C01796=1021.299,-78.040,-94.808,166.122,50.338,159.080
C01797=1021.304,-77.790,-94.818,166.125,50.334,159.080
C01798=1021.309,-77.541,-94.828,166.128,50.330,159.079
C01799=1021.315,-77.291,-94.838,166.131,50.326,159.079
C01800=1021.321,-77.042,-94.848,166.134,50.322,159.079
C01801=1021.326,-76.792,-94.858,166.137,50.318,159.079
C01802=1021.332,-76.542,-94.869,166.141,50.313,159.078
C01803=1021.337,-76.292,-94.879,166.143,50.309,159.078
C01804=1021.343,-76.042,-94.889,166.146,50.306,159.078
C01805=1021.349,-75.793,-94.899,166.149,50.302,159.078
C01806=1021.354,-75.543,-94.909,166.153,50.297,159.078
C01807=1021.360,-75.293,-94.920,166.155,50.293,159.077
C01808=1021.365,-75.044,-94.930,166.158,50.289,159.077
C01809=1021.371,-74.794,-94.940,166.162,50.285,159.077
C01810=1021.377,-74.544,-94.951,166.164,50.280,159.077
C01811=1021.383,-74.294,-94.961,166.167,50.276,159.076
C01812=1021.388,-74.045,-94.972,166.170,50.273,159.076
C01813=1021.394,-73.795,-94.982,166.174,50.269,159.076
C01814=1021.400,-73.545,-94.993,166.177,50.265,159.076
C01815=1021.405,-73.295,-95.003,166.180,50.261,159.076
C01816=1021.410,-73.046,-95.014,166.182,50.257,159.076
C01817=1021.416,-72.796,-95.024,166.185,50.253,159.075
C01818=1021.423,-72.475,-95.038,166.189,50.248,159.075
C01819=1021.430,-72.155,-95.051,166.193,50.243,159.075
C01820=1021.437,-71.835,-95.065,166.198,50.238,159.075
C01821=1021.444,-71.515,-95.079,166.201,50.233,159.074
C01822=1021.449,-71.265,-95.090,166.204,50.228,159.074
C01823=1021.454,-71.015,-95.100,166.207,50.225,159.074
C01824=1021.460,-70.766,-95.111,166.210,50.221,159.074
C01825=1021.466,-70.516,-95.122,166.213,50.217,159.073
C01826=1021.471,-70.286,-95.131,166.216,50.213,159.073
C01827=1021.476,-70.056,-95.141,166.219,50.209,159.073
C01828=1021.481,-69.826,-95.151,166.221,50.206,159.073
C01829=1021.487,-69.597,-95.161,166.224,50.202,159.073
C01830=1021.492,-69.367,-95.171,166.227,50.199,159.072
C01831=1021.497,-69.138,-95.180,166.229,50.195,159.072
C01832=1021.502,-68.907,-95.191,166.232,50.191,159.072
C01833=1021.507,-68.677,-95.200,166.235,50.187,159.072
C01834=1021.513,-68.428,-95.211,166.238,50.184,159.072
C01835=1021.518,-68.178,-95.222,166.241,50.180,159.071
C01836=1021.524,-67.928,-95.232,166.243,50.176,159.071
C01837=1021.530,-67.679,-95.243,166.247,50.171,159.071
C01838=1021.535,-67.429,-95.254,166.250,50.167,159.071
C01839=1021.541,-67.180,-95.265,166.253,50.164,159.071
C01840=1021.546,-66.930,-95.275,166.256,50.160,159.070
C01841=1021.552,-66.680,-95.286,166.259,50.155,159.070
C01842=1021.558,-66.431,-95.297,166.262,50.151,159.070
C01843=1021.564,-66.181,-95.308,166.265,50.147,159.070
C01844=1021.569,-65.932,-95.319,166.268,50.144,159.070
C01845=1021.575,-65.681,-95.330,166.272,50.139,159.069
C01846=1021.580,-65.431,-95.341,166.274,50.135,159.069
C01847=1021.586,-65.182,-95.352,166.277,50.131,159.069
C01848=1021.592,-64.932,-95.362,166.280,50.127,159.069
C01849=1021.598,-64.683,-95.373,166.282,50.123,159.068
C01850=1021.603,-64.433,-95.383,166.286,50.119,159.068
C01851=1021.609,-64.183,-95.394,166.289,50.115,159.068
C01852=1021.615,-63.934,-95.405,166.292,50.111,159.068
C01853=1021.620,-63.684,-95.416,166.294,50.107,159.067
C01854=1021.626,-63.434,-95.428,166.298,50.103,159.067
C01855=1021.632,-63.184,-95.439,166.301,50.099,159.067
C01856=1021.637,-62.935,-95.450,166.304,50.095,159.067
C01857=1021.643,-62.685,-95.461,166.306,50.090,159.066
C01858=1021.649,-62.436,-95.471,166.310,50.086,159.066
C01859=1021.654,-62.186,-95.482,166.313,50.083,159.066
C01860=1021.660,-61.936,-95.492,166.316,50.079,159.066
C01861=1021.666,-61.686,-95.504,166.318,50.075,159.066
C01862=1021.672,-61.436,-95.515,166.322,50.070,159.065
C01863=1021.677,-61.187,-95.526,166.325,50.066,159.065
C01864=1021.683,-60.937,-95.537,166.328,50.062,159.065
C01865=1021.689,-60.688,-95.548,166.330,50.058,159.064
C01866=1021.695,-60.437,-95.559,166.334,50.054,159.064
C01867=1021.701,-60.188,-95.570,166.337,50.050,159.064
C01868=1021.706,-59.938,-95.581,166.339,50.045,159.064
///RCONF 1,0,0,0,0,0,0,0,0,0,0,0,0,0,0,0,0,0,0,0,0,0,0,0
C01869=1021.712,-59.689,-95.592,166.343,50.041,159.064
C01870=1021.718,-59.439,-95.603,166.346,50.037,159.063
C01871=1021.724,-59.189,-95.614,166.349,50.033,159.063
C01872=1021.729,-58.939,-95.625,166.352,50.030,159.063
C01873=1021.735,-58.690,-95.636,166.355,50.025,159.063
C01874=1021.741,-58.441,-95.647,166.358,50.021,159.062
C01875=1021.747,-58.190,-95.658,166.361,50.017,159.062
C01876=1021.753,-57.941,-95.669,166.363,50.013,159.062
C01877=1021.759,-57.691,-95.680,166.367,50.009,159.062
C01878=1021.764,-57.442,-95.691,166.370,50.005,159.061
C01879=1021.770,-57.191,-95.703,166.373,50.000,159.061
C01880=1021.776,-56.942,-95.714,166.375,49.996,159.061
C01881=1021.782,-56.693,-95.725,166.379,49.992,159.061
C01882=1021.788,-56.443,-95.736,166.382,49.988,159.060
C01883=1021.794,-56.193,-95.747,166.384,49.984,159.060
C01884=1021.799,-55.944,-95.758,166.388,49.980,159.060
C01885=1021.804,-55.694,-95.770,166.391,49.975,159.060
C01886=1021.811,-55.444,-95.781,166.394,49.971,159.059
C01887=1021.817,-55.194,-95.792,166.396,49.967,159.059
C01888=1021.822,-54.945,-95.803,166.400,49.963,159.059
C01889=1021.829,-54.695,-95.815,166.403,49.959,159.059
C01890=1021.835,-54.446,-95.826,166.405,49.955,159.058
C01891=1021.840,-54.196,-95.836,166.409,49.950,159.058
C01892=1021.846,-53.946,-95.848,166.412,49.946,159.058
C01893=1021.852,-53.696,-95.859,166.414,49.942,159.057
C01894=1021.859,-53.417,-95.872,166.418,49.937,159.057
C01895=1021.866,-53.138,-95.884,166.421,49.932,159.057
C01896=1021.872,-52.859,-95.897,166.424,49.928,159.057
C01897=1021.879,-52.579,-95.909,166.427,49.923,159.056
C01898=1021.885,-52.330,-95.921,166.431,49.919,159.056
C01899=1021.890,-52.080,-95.932,166.434,49.915,159.056
C01900=1021.897,-51.830,-95.943,166.437,49.911,159.055
C01901=1021.902,-51.580,-95.955,166.439,49.907,159.055
C01902=1021.908,-51.331,-95.967,166.443,49.902,159.055
C01903=1021.914,-51.081,-95.977,166.446,49.898,159.055
C01904=1021.920,-50.832,-95.988,166.448,49.894,159.054
C01905=1021.926,-50.582,-96.001,166.451,49.890,159.054
C01906=1021.932,-50.332,-96.012,166.455,49.886,159.054
C01907=1021.937,-50.082,-96.024,166.458,49.882,159.054
C01908=1021.943,-49.833,-96.035,166.460,49.878,159.053
C01909=1021.949,-49.583,-96.047,166.463,49.874,159.053
C01910=1021.955,-49.334,-96.059,166.466,49.870,159.053
C01911=1021.960,-49.084,-96.070,166.469,49.866,159.053
C01912=1021.966,-48.834,-96.083,166.473,49.862,159.052
C01913=1021.971,-48.584,-96.094,166.475,49.858,159.052
C01914=1021.977,-48.335,-96.106,166.478,49.854,159.052
C01915=1021.983,-48.085,-96.117,166.481,49.850,159.052
C01916=1021.989,-47.835,-96.130,166.484,49.846,159.051
C01917=1021.995,-47.586,-96.140,166.486,49.842,159.051
C01918=1022.000,-47.337,-96.153,166.490,49.838,159.051
C01919=1022.006,-47.086,-96.164,166.493,49.834,159.051
C01920=1022.012,-46.837,-96.176,166.496,49.830,159.050
C01921=1022.017,-46.587,-96.188,166.498,49.826,159.050
C01922=1022.023,-46.338,-96.199,166.501,49.822,159.050
C01923=1022.029,-46.088,-96.212,166.504,49.818,159.050
C01924=1022.035,-45.838,-96.223,166.508,49.814,159.050
C01925=1022.041,-45.589,-96.235,166.511,49.810,159.049
C01926=1022.047,-45.339,-96.246,166.513,49.806,159.049
C01927=1022.053,-45.089,-96.259,166.516,49.802,159.049
C01928=1022.059,-44.840,-96.270,166.519,49.798,159.048
C01929=1022.064,-44.590,-96.282,166.521,49.794,159.048
C01930=1022.070,-44.341,-96.295,166.525,49.789,159.048
C01931=1022.076,-44.090,-96.306,166.528,49.785,159.048
C01932=1022.081,-43.841,-96.318,166.531,49.781,159.047
C01933=1022.088,-43.592,-96.330,166.533,49.777,159.047
C01934=1022.093,-43.341,-96.342,166.536,49.773,159.047
C01935=1022.099,-43.092,-96.353,166.540,49.770,159.047
C01936=1022.105,-42.842,-96.366,166.543,49.766,159.046
C01937=1022.110,-42.593,-96.377,166.546,49.762,159.046
C01938=1022.117,-42.343,-96.389,166.548,49.758,159.046
C01939=1022.122,-42.094,-96.401,166.551,49.753,159.045
C01940=1022.129,-41.844,-96.413,166.554,49.749,159.045
C01941=1022.134,-41.594,-96.425,166.558,49.745,159.045
C01942=1022.140,-41.345,-96.437,166.560,49.741,159.045
C01943=1022.147,-41.095,-96.449,166.563,49.737,159.044
C01944=1022.152,-40.845,-96.461,166.566,49.733,159.044
C01945=1022.158,-40.596,-96.473,166.568,49.729,159.044
C01946=1022.163,-40.346,-96.485,166.572,49.725,159.044
C01947=1022.170,-40.097,-96.497,166.575,49.721,159.043
C01948=1022.176,-39.846,-96.509,166.578,49.717,159.043
C01949=1022.181,-39.597,-96.521,166.580,49.713,159.043
C01950=1022.188,-39.348,-96.533,166.583,49.708,159.042
C01951=1022.194,-39.098,-96.546,166.587,49.704,159.042
C01952=1022.199,-38.849,-96.558,166.589,49.700,159.042
C01953=1022.204,-38.598,-96.570,166.592,49.696,159.042
C01954=1022.210,-38.348,-96.582,166.595,49.692,159.041
C01955=1022.216,-38.099,-96.594,166.598,49.688,159.041
C01956=1022.222,-37.849,-96.606,166.601,49.685,159.041
C01957=1022.228,-37.600,-96.619,166.603,49.681,159.041
C01958=1022.234,-37.321,-96.633,166.607,49.676,159.040
C01959=1022.241,-37.043,-96.646,166.610,49.672,159.040
C01960=1022.248,-36.763,-96.659,166.613,49.667,159.040
C01961=1022.253,-36.484,-96.673,166.617,49.662,159.039
C01962=1022.259,-36.234,-96.686,166.620,49.659,159.039
C01963=1022.265,-35.984,-96.699,166.623,49.655,159.039
C01964=1022.271,-35.735,-96.711,166.625,49.651,159.039
C01965=1022.277,-35.486,-96.723,166.628,49.647,159.038
C01966=1022.283,-35.236,-96.735,166.631,49.643,159.038
C01967=1022.288,-34.987,-96.747,166.633,49.639,159.038
C01968=1022.294,-34.737,-96.760,166.636,49.635,159.037
C01969=1022.300,-34.487,-96.773,166.640,49.630,159.037
C01970=1022.306,-34.237,-96.785,166.643,49.626,159.037
C01971=1022.312,-33.988,-96.797,166.645,49.622,159.037
C01972=1022.318,-33.738,-96.809,166.648,49.618,159.036
C01973=1022.324,-33.488,-96.822,166.651,49.615,159.036
C01974=1022.330,-33.238,-96.834,166.654,49.611,159.036
C01975=1022.336,-32.990,-96.847,166.657,49.607,159.036
C01976=1022.341,-32.740,-96.860,166.659,49.603,159.035
C01977=1022.347,-32.490,-96.872,166.663,49.599,159.035
C01978=1022.353,-32.240,-96.885,166.666,49.595,159.035
C01979=1022.359,-31.991,-96.897,166.669,49.591,159.035
C01980=1022.365,-31.742,-96.909,166.671,49.587,159.034
C01981=1022.371,-31.492,-96.922,166.674,49.583,159.034
C01982=1022.377,-31.242,-96.934,166.677,49.579,159.034
C01983=1022.382,-30.993,-96.946,166.679,49.575,159.033
C01984=1022.388,-30.743,-96.959,166.682,49.570,159.033
C01985=1022.395,-30.493,-96.972,166.686,49.566,159.033
C01986=1022.400,-30.244,-96.985,166.689,49.562,159.033
C01987=1022.406,-29.994,-96.997,166.691,49.558,159.032
C01988=1022.412,-29.745,-97.009,166.694,49.554,159.032
C01989=1022.418,-29.495,-97.021,166.697,49.550,159.032
C01990=1022.424,-29.245,-97.034,166.700,49.546,159.031
C01991=1022.430,-28.996,-97.047,166.702,49.542,159.031
C01992=1022.436,-28.746,-97.060,166.706,49.538,159.031
C01993=1022.442,-28.496,-97.072,166.709,49.534,159.031
C01994=1022.448,-28.247,-97.085,166.711,49.530,159.030
C01995=1022.453,-27.997,-97.097,166.714,49.526,159.030
C01996=1022.460,-27.748,-97.110,166.717,49.522,159.030
C01997=1022.466,-27.498,-97.122,166.720,49.518,159.029
C01998=1022.471,-27.248,-97.136,166.722,49.514,159.029
C01999=1022.477,-26.998,-97.148,166.725,49.510,159.029
C02000=1022.484,-26.749,-97.161,166.728,49.506,159.028
C02001=1022.489,-26.499,-97.174,166.731,49.502,159.028
C02002=1022.495,-26.250,-97.186,166.734,49.497,159.028
C02003=1022.501,-26.000,-97.199,166.737,49.493,159.028
C02004=1022.506,-25.750,-97.213,166.740,49.490,159.028
C02005=1022.512,-25.501,-97.226,166.743,49.486,159.027
C02006=1022.518,-25.251,-97.238,166.746,49.482,159.027
C02007=1022.524,-25.001,-97.251,166.748,49.478,159.027
C02008=1022.530,-24.752,-97.264,166.751,49.474,159.026
C02009=1022.536,-24.502,-97.277,166.754,49.470,159.026
C02010=1022.541,-24.253,-97.290,166.757,49.466,159.026
C02011=1022.547,-24.003,-97.303,166.759,49.462,159.025
C02012=1022.553,-23.754,-97.316,166.762,49.458,159.025
C02013=1022.559,-23.504,-97.329,166.765,49.454,159.025
C02014=1022.565,-23.255,-97.342,166.768,49.450,159.024
C02015=1022.571,-23.005,-97.354,166.770,49.446,159.024
C02016=1022.577,-22.755,-97.368,166.773,49.443,159.024
C02017=1022.583,-22.506,-97.381,166.776,49.439,159.024
C02018=1022.589,-22.256,-97.393,166.779,49.435,159.023
C02019=1022.595,-22.006,-97.407,166.783,49.430,159.023
C02020=1022.601,-21.756,-97.419,166.785,49.426,159.023
C02021=1022.606,-21.507,-97.433,166.788,49.422,159.023
C02022=1022.613,-21.228,-97.447,166.790,49.418,159.022
C02023=1022.620,-20.947,-97.462,166.794,49.413,159.022
C02024=1022.626,-20.668,-97.477,166.797,49.409,159.021
C02025=1022.633,-20.388,-97.491,166.800,49.404,159.021
C02026=1022.639,-20.138,-97.504,166.803,49.400,159.021
C02027=1022.645,-19.889,-97.517,166.806,49.396,159.021
C02028=1022.651,-19.639,-97.530,166.809,49.392,159.020
C02029=1022.657,-19.389,-97.544,166.811,49.388,159.020
C02030=1022.663,-19.140,-97.556,166.814,49.384,159.020
C02031=1022.669,-18.890,-97.570,166.817,49.380,159.019
C02032=1022.675,-18.641,-97.583,166.820,49.376,159.019
C02033=1022.680,-18.391,-97.596,166.823,49.372,159.019
C02034=1022.687,-18.142,-97.609,166.826,49.368,159.019
C02035=1022.693,-17.892,-97.622,166.829,49.364,159.018
C02036=1022.699,-17.642,-97.635,166.832,49.360,159.018
C02037=1022.705,-17.393,-97.648,166.834,49.356,159.018
C02038=1022.711,-17.143,-97.661,166.837,49.352,159.017
C02039=1022.716,-16.894,-97.675,166.840,49.348,159.017
C02040=1022.722,-16.644,-97.688,166.842,49.343,159.017
C02041=1022.728,-16.395,-97.701,166.845,49.339,159.016
C02042=1022.735,-16.145,-97.714,166.848,49.335,159.016
C02043=1022.741,-15.896,-97.727,166.850,49.331,159.016
C02044=1022.746,-15.646,-97.740,166.853,49.327,159.015
C02045=1022.752,-15.397,-97.753,166.856,49.323,159.015
C02046=1022.758,-15.147,-97.767,166.859,49.319,159.015
C02047=1022.764,-14.898,-97.781,166.862,49.316,159.015
C02048=1022.769,-14.648,-97.794,166.864,49.312,159.014
C02049=1022.776,-14.398,-97.807,166.867,49.308,159.014
C02050=1022.781,-14.148,-97.821,166.870,49.304,159.014
C02051=1022.788,-13.899,-97.835,166.873,49.300,159.013
C02052=1022.793,-13.649,-97.848,166.875,49.296,159.013
C02053=1022.799,-13.400,-97.862,166.878,49.292,159.013
C02054=1022.805,-13.151,-97.875,166.881,49.288,159.012
C02055=1022.811,-12.900,-97.888,166.884,49.284,159.012
C02056=1022.817,-12.651,-97.901,166.886,49.280,159.012
C02057=1022.822,-12.402,-97.915,166.889,49.276,159.011
C02058=1022.829,-12.152,-97.928,166.892,49.272,159.011
C02059=1022.835,-11.902,-97.943,166.895,49.268,159.011
C02060=1022.841,-11.653,-97.956,166.897,49.264,159.010
C02061=1022.846,-11.403,-97.970,166.900,49.260,159.010
C02062=1022.853,-11.154,-97.983,166.903,49.256,159.010
C02063=1022.858,-10.904,-97.997,166.906,49.252,159.010
C02064=1022.864,-10.655,-98.010,166.908,49.248,159.009
C02065=1022.869,-10.405,-98.023,166.911,49.244,159.009
C02066=1022.876,-10.155,-98.037,166.915,49.240,159.009
C02067=1022.882,-9.905,-98.051,166.918,49.236,159.008
C02068=1022.888,-9.656,-98.064,166.920,49.232,159.008
C02069=1022.893,-9.406,-98.078,166.923,49.228,159.008
C02070=1022.900,-9.157,-98.091,166.926,49.224,159.007
C02071=1022.905,-8.908,-98.105,166.929,49.220,159.007
C02072=1022.912,-8.658,-98.119,166.931,49.216,159.007
C02073=1022.918,-8.408,-98.132,166.934,49.212,159.007
C02074=1022.924,-8.159,-98.146,166.937,49.208,159.006
C02075=1022.930,-7.910,-98.159,166.940,49.204,159.006
C02076=1022.935,-7.660,-98.173,166.942,49.200,159.006
C02077=1022.942,-7.410,-98.187,166.945,49.196,159.005
C02078=1022.948,-7.160,-98.201,166.948,49.192,159.005
C02079=1022.954,-6.911,-98.214,166.951,49.188,159.005
C02080=1022.959,-6.662,-98.228,166.953,49.184,159.004
C02081=1022.966,-6.412,-98.241,166.956,49.180,159.004
C02082=1022.972,-6.162,-98.255,166.959,49.176,159.004
C02083=1022.978,-5.913,-98.268,166.962,49.172,159.003
C02084=1022.983,-5.663,-98.282,166.964,49.169,159.003
C02085=1022.990,-5.414,-98.297,166.967,49.165,159.003
C02086=1022.997,-5.132,-98.312,166.970,49.160,159.002
C02087=1023.003,-4.851,-98.328,166.973,49.155,159.002
C02088=1023.010,-4.569,-98.343,166.977,49.151,159.002
C02089=1023.017,-4.288,-98.359,166.979,49.146,159.001
C02090=1023.023,-4.039,-98.372,166.982,49.142,159.001
C02091=1023.029,-3.788,-98.386,166.985,49.138,159.001
C02092=1023.034,-3.539,-98.400,166.987,49.134,159.000
C02093=1023.040,-3.289,-98.414,166.990,49.130,159.000
C02094=1023.046,-3.040,-98.429,166.993,49.127,159.000
C02095=1023.052,-2.790,-98.443,166.996,49.123,158.999
C02096=1023.058,-2.541,-98.456,166.999,49.119,158.999
C02097=1023.064,-2.292,-98.471,167.002,49.115,158.999
C02098=1023.070,-2.041,-98.485,167.003,49.111,158.998
C02099=1023.075,-1.792,-98.499,167.006,49.107,158.998
C02100=1023.081,-1.543,-98.513,167.009,49.103,158.998
C02101=1023.087,-1.293,-98.528,167.012,49.099,158.997
C02102=1023.093,-1.043,-98.541,167.014,49.095,158.997
C02103=1023.099,-0.794,-98.555,167.017,49.091,158.997
C02104=1023.105,-0.545,-98.569,167.020,49.087,158.997
C02105=1023.111,-0.295,-98.584,167.023,49.083,158.996
C02106=1023.117,-0.046,-98.598,167.026,49.080,158.996
C02107=1023.122,0.204,-98.612,167.028,49.076,158.996
C02108=1023.128,0.454,-98.626,167.031,49.072,158.995
C02109=1023.134,0.703,-98.641,167.034,49.068,158.995
C02110=1023.140,0.952,-98.654,167.037,49.064,158.995
C02111=1023.146,1.203,-98.668,167.039,49.060,158.994
C02112=1023.152,1.452,-98.683,167.041,49.057,158.994
C02113=1023.157,1.701,-98.697,167.044,49.053,158.994
C02114=1023.164,1.951,-98.712,167.047,49.049,158.993
C02115=1023.169,2.200,-98.726,167.049,49.045,158.993
C02116=1023.176,2.450,-98.741,167.052,49.041,158.993
C02117=1023.182,2.699,-98.754,167.055,49.037,158.992
C02118=1023.187,2.949,-98.768,167.058,49.033,158.992
C02119=1023.194,3.199,-98.783,167.060,49.029,158.992
C02120=1023.199,3.448,-98.796,167.063,49.025,158.991
C02121=1023.205,3.697,-98.811,167.066,49.021,158.991
C02122=1023.211,3.947,-98.825,167.069,49.017,158.991
C02123=1023.217,4.196,-98.840,167.072,49.013,158.991
C02124=1023.223,4.447,-98.854,167.074,49.009,158.990
C02125=1023.229,4.695,-98.868,167.077,49.005,158.990
C02126=1023.236,4.946,-98.882,167.080,49.001,158.990
C02127=1023.241,5.195,-98.897,167.083,48.997,158.989
C02128=1023.247,5.444,-98.911,167.084,48.994,158.989
C02129=1023.253,5.694,-98.926,167.087,48.990,158.989
C02130=1023.259,5.943,-98.940,167.089,48.985,158.988
C02131=1023.265,6.193,-98.954,167.092,48.981,158.988
C02132=1023.271,6.443,-98.968,167.095,48.977,158.987
C02133=1023.278,6.692,-98.983,167.098,48.973,158.987
C02134=1023.283,6.941,-98.997,167.101,48.969,158.987
C02135=1023.289,7.190,-99.011,167.103,48.965,158.986
C02136=1023.295,7.440,-99.026,167.106,48.961,158.986
C02137=1023.301,7.690,-99.040,167.109,48.957,158.986
C02138=1023.307,7.939,-99.055,167.112,48.953,158.985
C02139=1023.313,8.189,-99.069,167.114,48.950,158.985
C02140=1023.319,8.439,-99.084,167.117,48.946,158.985
C02141=1023.325,8.688,-99.098,167.120,48.941,158.984
C02142=1023.332,8.937,-99.112,167.122,48.937,158.984
C02143=1023.337,9.186,-99.127,167.125,48.933,158.984
C02144=1023.343,9.437,-99.141,167.128,48.929,158.983
C02145=1023.349,9.686,-99.155,167.131,48.925,158.983
C02146=1023.356,9.935,-99.170,167.133,48.921,158.983
C02147=1023.361,10.185,-99.184,167.136,48.917,158.982
C02148=1023.367,10.435,-99.199,167.139,48.913,158.982
C02149=1023.373,10.684,-99.214,167.141,48.909,158.982
C02150=1023.380,10.967,-99.230,167.144,48.905,158.981
C02151=1023.387,11.250,-99.246,167.148,48.900,158.981
C02152=1023.394,11.534,-99.263,167.150,48.895,158.980
C02153=1023.402,11.817,-99.279,167.153,48.890,158.980
C02154=1023.407,12.066,-99.294,167.156,48.886,158.980
C02155=1023.413,12.317,-99.308,167.159,48.882,158.979
C02156=1023.420,12.566,-99.323,167.162,48.878,158.979
C02157=1023.426,12.815,-99.337,167.164,48.875,158.979
C02158=1023.432,13.066,-99.352,167.166,48.871,158.978
C02159=1023.437,13.314,-99.366,167.169,48.866,158.978
C02160=1023.444,13.564,-99.381,167.172,48.862,158.977
C02161=1023.450,13.814,-99.396,167.174,48.858,158.977
C02162=1023.456,14.063,-99.411,167.177,48.854,158.977
C02163=1023.462,14.313,-99.425,167.180,48.850,158.976
C02164=1023.467,14.562,-99.440,167.183,48.846,158.976
C02165=1023.473,14.812,-99.455,167.185,48.843,158.976
C02166=1023.479,15.061,-99.470,167.188,48.839,158.975
C02167=1023.486,15.311,-99.485,167.191,48.835,158.975
C02168=1023.492,15.560,-99.500,167.194,48.831,158.975
C02169=1023.498,15.809,-99.514,167.195,48.827,158.974
C02170=1023.503,16.059,-99.530,167.198,48.823,158.974
C02171=1023.509,16.308,-99.544,167.201,48.819,158.974
C02172=1023.515,16.558,-99.558,167.204,48.815,158.973
C02173=1023.522,16.808,-99.573,167.207,48.811,158.973
C02174=1023.527,17.057,-99.588,167.209,48.807,158.973
C02175=1023.533,17.307,-99.604,167.212,48.803,158.972
C02176=1023.539,17.556,-99.618,167.215,48.799,158.972
C02177=1023.545,17.806,-99.633,167.217,48.795,158.972
C02178=1023.552,18.055,-99.648,167.220,48.791,158.971
C02179=1023.557,18.304,-99.663,167.222,48.787,158.971
C02180=1023.563,18.554,-99.678,167.225,48.783,158.971
C02181=1023.569,18.804,-99.693,167.227,48.779,158.970
C02182=1023.575,19.053,-99.708,167.230,48.776,158.970
C02183=1023.582,19.302,-99.723,167.233,48.772,158.970
C02184=1023.588,19.552,-99.738,167.236,48.768,158.969
C02185=1023.593,19.801,-99.753,167.238,48.763,158.969
C02186=1023.599,20.051,-99.768,167.241,48.759,158.968
C02187=1023.606,20.301,-99.783,167.243,48.755,158.968
C02188=1023.611,20.550,-99.798,167.245,48.752,158.968
C02189=1023.617,20.800,-99.813,167.248,48.748,158.967
C02190=1023.624,21.049,-99.828,167.251,48.744,158.967
C02191=1023.629,21.298,-99.844,167.254,48.740,158.967
C02192=1023.635,21.548,-99.858,167.257,48.736,158.966
C02193=1023.642,21.797,-99.873,167.259,48.732,158.966
C02194=1023.647,22.046,-99.889,167.262,48.728,158.966
C02195=1023.653,22.296,-99.904,167.264,48.724,158.965
C02196=1023.659,22.546,-99.919,167.267,48.720,158.965
C02197=1023.665,22.795,-99.934,167.269,48.716,158.965
C02198=1023.671,23.044,-99.949,167.272,48.713,158.964
C02199=1023.677,23.294,-99.965,167.275,48.708,158.964
C02200=1023.683,23.544,-99.980,167.277,48.704,158.963
C02201=1023.689,23.793,-99.994,167.280,48.700,158.963
C02202=1023.695,24.043,-100.010,167.283,48.696,158.963
C02203=1023.701,24.292,-100.025,167.285,48.693,158.962
C02204=1023.707,24.541,-100.040,167.288,48.689,158.962
C02205=1023.713,24.791,-100.056,167.290,48.685,158.962
C02206=1023.719,25.040,-100.071,167.293,48.681,158.961
C02207=1023.726,25.290,-100.086,167.296,48.676,158.961
C02208=1023.731,25.539,-100.101,167.298,48.672,158.961
C02209=1023.737,25.788,-100.116,167.301,48.668,158.960
C02210=1023.743,26.038,-100.132,167.304,48.664,158.960
C02211=1023.749,26.288,-100.147,167.307,48.661,158.960
C02212=1023.755,26.537,-100.162,167.308,48.657,158.959
C02213=1023.761,26.786,-100.178,167.311,48.653,158.959
C02214=1023.768,27.071,-100.195,167.315,48.648,158.958
C02215=1023.775,27.356,-100.212,167.317,48.643,158.958
C02216=1023.782,27.641,-100.230,167.321,48.639,158.958
C02217=1023.788,27.926,-100.247,167.323,48.635,158.957
C02218=1023.795,28.175,-100.263,167.326,48.631,158.957
C02219=1023.801,28.425,-100.278,167.329,48.627,158.956
C02220=1023.806,28.675,-100.294,167.331,48.623,158.956
C02221=1023.813,28.923,-100.309,167.334,48.619,158.956
C02222=1023.818,29.173,-100.325,167.336,48.615,158.955
C02223=1023.825,29.422,-100.341,167.339,48.611,158.955
C02224=1023.831,29.672,-100.356,167.342,48.608,158.955
C02225=1023.836,29.922,-100.372,167.344,48.603,158.954
C02226=1023.842,30.170,-100.387,167.346,48.599,158.954
C02227=1023.848,30.420,-100.402,167.349,48.595,158.953
C02228=1023.855,30.669,-100.418,167.352,48.591,158.953
C02229=1023.860,30.919,-100.434,167.355,48.588,158.953
C02230=1023.866,31.169,-100.450,167.357,48.584,158.952
C02231=1023.873,31.418,-100.465,167.360,48.580,158.952
C02232=1023.878,31.667,-100.481,167.362,48.576,158.952
C02233=1023.884,31.917,-100.496,167.365,48.572,158.951
C02234=1023.890,32.166,-100.512,167.367,48.568,158.951
C02235=1023.896,32.416,-100.527,167.370,48.564,158.951
C02236=1023.903,32.665,-100.543,167.373,48.560,158.950
C02237=1023.908,32.915,-100.559,167.375,48.556,158.950
C02238=1023.914,33.163,-100.574,167.378,48.552,158.950
C02239=1023.920,33.413,-100.590,167.380,48.548,158.949
C02240=1023.926,33.663,-100.606,167.383,48.544,158.949
C02241=1023.932,33.912,-100.621,167.386,48.541,158.948
C02242=1023.938,34.162,-100.637,167.388,48.537,158.948
C02243=1023.944,34.412,-100.653,167.391,48.532,158.948
C02244=1023.951,34.661,-100.668,167.394,48.528,158.947
C02245=1023.956,34.911,-100.684,167.395,48.525,158.947
C02246=1023.963,35.160,-100.699,167.398,48.521,158.946
C02247=1023.968,35.409,-100.715,167.401,48.517,158.946
C02248=1023.974,35.658,-100.731,167.404,48.513,158.946
C02249=1023.981,35.907,-100.746,167.406,48.508,158.945
C02250=1023.986,36.157,-100.762,167.409,48.504,158.945
C02251=1023.993,36.406,-100.778,167.412,48.500,158.945
C02252=1023.999,36.656,-100.793,167.415,48.497,158.944
C02253=1024.005,36.906,-100.809,167.416,48.493,158.944
C02254=1024.010,37.155,-100.826,167.419,48.489,158.944
C02255=1024.017,37.405,-100.841,167.422,48.485,158.943
C02256=1024.023,37.654,-100.857,167.425,48.481,158.943
C02257=1024.029,37.903,-100.873,167.428,48.477,158.943
C02258=1024.034,38.153,-100.889,167.429,48.473,158.942
C02259=1024.040,38.402,-100.905,167.432,48.469,158.942
C02260=1024.046,38.651,-100.921,167.435,48.465,158.941
C02261=1024.052,38.901,-100.937,167.437,48.461,158.941
C02262=1024.058,39.150,-100.952,167.440,48.457,158.941
C02263=1024.064,39.400,-100.968,167.442,48.454,158.940
C02264=1024.070,39.649,-100.985,167.445,48.450,158.940
C02265=1024.076,39.898,-101.001,167.448,48.446,158.940
C02266=1024.082,40.148,-101.017,167.450,48.442,158.939
C02267=1024.087,40.398,-101.033,167.453,48.438,158.939
C02268=1024.093,40.647,-101.049,167.455,48.435,158.938
C02269=1024.100,40.896,-101.065,167.457,48.430,158.938
C02270=1024.106,41.145,-101.081,167.460,48.426,158.938
C02271=1024.112,41.395,-101.096,167.463,48.422,158.937
C02272=1024.118,41.645,-101.113,167.466,48.418,158.937
C02273=1024.124,41.894,-101.129,167.469,48.415,158.937
C02274=1024.130,42.143,-101.145,167.470,48.411,158.936
C02275=1024.136,42.393,-101.161,167.473,48.407,158.936
C02276=1024.141,42.642,-101.178,167.476,48.403,158.935
C02277=1024.147,42.891,-101.194,167.479,48.399,158.935
C02278=1024.154,43.176,-101.212,167.481,48.395,158.935
C02279=1024.161,43.461,-101.231,167.484,48.391,158.934
C02280=1024.168,43.747,-101.249,167.488,48.386,158.934
C02281=1024.174,44.031,-101.268,167.490,48.381,158.933
C02282=1024.180,44.280,-101.284,167.493,48.377,158.933
C02283=1024.186,44.530,-101.300,167.495,48.374,158.933
C02284=1024.192,44.779,-101.316,167.498,48.370,158.932
C02285=1024.197,45.029,-101.333,167.500,48.366,158.932
C02286=1024.203,45.278,-101.350,167.503,48.362,158.932
C02287=1024.209,45.527,-101.366,167.505,48.359,158.931
C02288=1024.215,45.777,-101.382,167.508,48.355,158.931
C02289=1024.221,46.026,-101.398,167.511,48.351,158.930
C02290=1024.227,46.275,-101.415,167.513,48.347,158.930
C02291=1024.233,46.525,-101.431,167.515,48.343,158.930
C02292=1024.238,46.774,-101.448,167.518,48.339,158.929
C02293=1024.244,47.024,-101.464,167.521,48.336,158.929
C02294=1024.250,47.272,-101.481,167.524,48.332,158.929
C02295=1024.256,47.522,-101.497,167.525,48.328,158.928
C02296=1024.262,47.771,-101.513,167.528,48.324,158.928
C02297=1024.269,48.021,-101.530,167.531,48.320,158.928
C02298=1024.274,48.271,-101.547,167.534,48.317,158.927
C02299=1024.280,48.520,-101.563,167.535,48.313,158.927
C02300=1024.286,48.770,-101.579,167.538,48.309,158.926
C02301=1024.292,49.019,-101.596,167.541,48.305,158.926
C02302=1024.298,49.268,-101.612,167.544,48.301,158.926
C02303=1024.304,49.518,-101.628,167.547,48.297,158.925
C02304=1024.310,49.766,-101.645,167.549,48.294,158.925
C02305=1024.315,50.016,-101.662,167.551,48.289,158.924
C02306=1024.321,50.265,-101.678,167.554,48.285,158.924
C02307=1024.327,50.515,-101.695,167.557,48.281,158.924
C02308=1024.333,50.764,-101.711,167.558,48.278,158.923
C02309=1024.340,51.014,-101.727,167.561,48.274,158.923
C02310=1024.345,51.263,-101.744,167.564,48.270,158.923
C02311=1024.351,51.512,-101.761,167.567,48.266,158.922
C02312=1024.357,51.762,-101.778,167.570,48.262,158.922
C02313=1024.363,52.011,-101.794,167.571,48.259,158.922
C02314=1024.369,52.261,-101.810,167.574,48.254,158.921
C02315=1024.375,52.510,-101.826,167.577,48.250,158.921
C02316=1024.382,52.759,-101.844,167.580,48.247,158.920
C02317=1024.387,53.009,-101.860,167.582,48.243,158.920
C02318=1024.393,53.258,-101.877,167.584,48.239,158.920
C02319=1024.399,53.508,-101.893,167.587,48.235,158.919
C02320=1024.405,53.757,-101.909,167.589,48.231,158.919
C02321=1024.411,54.006,-101.926,167.592,48.227,158.918
C02322=1024.417,54.256,-101.943,167.595,48.223,158.918
C02323=1024.423,54.505,-101.960,167.597,48.219,158.918
C02324=1024.429,54.755,-101.976,167.600,48.215,158.917
C02325=1024.435,55.004,-101.993,167.602,48.212,158.917
C02326=1024.441,55.253,-102.009,167.605,48.207,158.916
C02327=1024.447,55.502,-102.025,167.608,48.203,158.916
C02328=1024.453,55.752,-102.043,167.610,48.200,158.916
C02329=1024.459,56.001,-102.060,167.612,48.196,158.915
C02330=1024.465,56.251,-102.076,167.615,48.192,158.915
C02331=1024.471,56.500,-102.092,167.618,48.187,158.914
C02332=1024.477,56.749,-102.109,167.621,48.183,158.914
C02333=1024.483,56.999,-102.126,167.623,48.180,158.914
C02334=1024.489,57.248,-102.143,167.625,48.176,158.913
C02335=1024.495,57.497,-102.160,167.628,48.172,158.913
C02336=1024.501,57.747,-102.176,167.630,48.168,158.912
C02337=1024.508,57.997,-102.192,167.633,48.164,158.912
C02338=1024.514,58.245,-102.209,167.636,48.160,158.912
C02339=1024.519,58.495,-102.226,167.638,48.156,158.911
C02340=1024.525,58.744,-102.242,167.640,48.152,158.911
C02341=1024.532,58.994,-102.260,167.643,48.148,158.911
C02342=1024.538,59.278,-102.278,167.647,48.143,158.910
C02343=1024.545,59.563,-102.297,167.649,48.138,158.910
C02344=1024.553,59.847,-102.317,167.652,48.134,158.909
C02345=1024.559,60.131,-102.336,167.656,48.130,158.909
C02346=1024.565,60.382,-102.353,167.658,48.125,158.908
C02347=1024.571,60.630,-102.370,167.660,48.122,158.908
C02348=1024.577,60.880,-102.386,167.663,48.118,158.907
C02349=1024.584,61.130,-102.403,167.665,48.113,158.907
C02350=1024.590,61.379,-102.420,167.668,48.109,158.907
C02351=1024.595,61.628,-102.437,167.671,48.106,158.906
C02352=1024.602,61.877,-102.454,167.674,48.102,158.906
C02353=1024.608,62.127,-102.470,167.675,48.097,158.905
C02354=1024.615,62.376,-102.487,167.678,48.094,158.905
C02355=1024.620,62.625,-102.503,167.681,48.090,158.905
C02356=1024.627,62.875,-102.521,167.683,48.085,158.904
C02357=1024.633,63.124,-102.538,167.686,48.081,158.904
C02358=1024.639,63.373,-102.555,167.689,48.078,158.903
C02359=1024.645,63.623,-102.572,167.691,48.074,158.903
C02360=1024.651,63.872,-102.589,167.694,48.070,158.903
C02361=1024.657,64.122,-102.606,167.696,48.066,158.902
C02362=1024.663,64.371,-102.623,167.699,48.062,158.902
C02363=1024.668,64.621,-102.640,167.702,48.058,158.901
C02364=1024.674,64.869,-102.657,167.703,48.054,158.901
C02365=1024.681,65.119,-102.675,167.706,48.050,158.901
C02366=1024.686,65.369,-102.691,167.709,48.047,158.900
C02367=1024.692,65.618,-102.709,167.712,48.042,158.900
C02368=1024.699,65.867,-102.726,167.714,48.038,158.899
C02369=1024.704,66.117,-102.743,167.716,48.035,158.899
C02370=1024.711,66.366,-102.760,167.719,48.031,158.899
C02371=1024.716,66.615,-102.778,167.722,48.027,158.898
C02372=1024.722,66.864,-102.794,167.725,48.023,158.898
C02373=1024.729,67.114,-102.812,167.726,48.019,158.897
C02374=1024.734,67.363,-102.829,167.729,48.015,158.897
C02375=1024.740,67.612,-102.846,167.732,48.011,158.897
C02376=1024.746,67.862,-102.864,167.735,48.007,158.896
C02377=1024.752,68.111,-102.881,167.738,48.003,158.896
C02378=1024.758,68.360,-102.898,167.739,48.000,158.896
C02379=1024.764,68.610,-102.915,167.742,47.995,158.895
C02380=1024.770,68.859,-102.932,167.745,47.992,158.895
C02381=1024.776,69.109,-102.950,167.748,47.988,158.894
C02382=1024.782,69.358,-102.967,167.749,47.984,158.894
C02383=1024.788,69.607,-102.985,167.752,47.980,158.894
C02384=1024.794,69.857,-103.002,167.755,47.976,158.893
C02385=1024.799,70.106,-103.020,167.758,47.973,158.893
C02386=1024.805,70.355,-103.037,167.761,47.969,158.893
C02387=1024.812,70.605,-103.055,167.762,47.965,158.892
C02388=1024.817,70.854,-103.072,167.765,47.961,158.892
C02389=1024.824,71.103,-103.089,167.768,47.957,158.891
C02390=1024.829,71.352,-103.107,167.771,47.953,158.891
C02391=1024.835,71.602,-103.124,167.772,47.949,158.890
C02392=1024.841,71.851,-103.142,167.775,47.946,158.890
C02393=1024.847,72.100,-103.159,167.778,47.942,158.890
C02394=1024.853,72.350,-103.177,167.781,47.938,158.889
C02395=1024.859,72.599,-103.194,167.782,47.934,158.889
C02396=1024.866,72.848,-103.212,167.785,47.930,158.888
C02397=1024.871,73.097,-103.229,167.788,47.926,158.888
C02398=1024.877,73.347,-103.247,167.791,47.922,158.888
C02399=1024.883,73.596,-103.265,167.794,47.918,158.887
C02400=1024.889,73.845,-103.282,167.796,47.915,158.887
C02401=1024.895,74.095,-103.300,167.798,47.910,158.886
C02402=1024.901,74.344,-103.317,167.801,47.906,158.886
C02403=1024.906,74.594,-103.334,167.804,47.903,158.886
C02404=1024.913,74.843,-103.351,167.806,47.899,158.885
C02405=1024.919,75.093,-103.369,167.808,47.895,158.885
C02406=1024.925,75.377,-103.390,167.812,47.890,158.884
C02407=1024.932,75.661,-103.410,167.814,47.886,158.884
C02408=1024.939,75.945,-103.429,167.817,47.881,158.883
C02409=1024.946,76.229,-103.450,167.821,47.877,158.883
C02410=1024.952,76.479,-103.468,167.822,47.873,158.883
C02411=1024.958,76.728,-103.486,167.825,47.869,158.882
C02412=1024.964,76.978,-103.503,167.828,47.865,158.882
C02413=1024.970,77.227,-103.521,167.831,47.862,158.882
C02414=1024.976,77.476,-103.539,167.833,47.858,158.881
C02415=1024.982,77.725,-103.556,167.836,47.854,158.881
C02416=1024.988,77.975,-103.574,167.838,47.850,158.880
C02417=1024.993,78.224,-103.592,167.841,47.847,158.880
C02418=1024.999,78.474,-103.610,167.843,47.843,158.880
C02419=1025.005,78.723,-103.627,167.846,47.839,158.879
C02420=1025.011,78.972,-103.646,167.848,47.835,158.879
C02421=1025.017,79.221,-103.663,167.851,47.831,158.878
C02422=1025.023,79.471,-103.681,167.853,47.827,158.878
C02423=1025.028,79.720,-103.699,167.856,47.823,158.878
C02424=1025.035,79.970,-103.717,167.859,47.820,158.877
C02425=1025.040,80.218,-103.735,167.862,47.816,158.877
C02426=1025.047,80.468,-103.753,167.863,47.812,158.876
C02427=1025.052,80.717,-103.771,167.866,47.808,158.876
C02428=1025.058,80.967,-103.788,167.869,47.805,158.876
C02429=1025.064,81.216,-103.806,167.872,47.801,158.875
C02430=1025.070,81.465,-103.825,167.873,47.797,158.875
C02431=1025.076,81.714,-103.842,167.876,47.793,158.874
C02432=1025.081,81.964,-103.861,167.879,47.789,158.874
C02433=1025.087,82.213,-103.878,167.882,47.785,158.874
C02434=1025.093,82.462,-103.897,167.885,47.781,158.873
C02435=1025.099,82.712,-103.915,167.887,47.778,158.873
C02436=1025.105,82.961,-103.933,167.889,47.774,158.873
C02437=1025.111,83.210,-103.950,167.892,47.770,158.872
C02438=1025.117,83.459,-103.969,167.895,47.766,158.872
C02439=1025.123,83.709,-103.987,167.897,47.762,158.871
C02440=1025.128,83.958,-104.004,167.899,47.758,158.871
C02441=1025.135,84.207,-104.023,167.902,47.755,158.871
C02442=1025.141,84.457,-104.041,167.905,47.751,158.870
C02443=1025.146,84.706,-104.058,167.908,47.747,158.870
C02444=1025.153,84.955,-104.077,167.910,47.743,158.869
C02445=1025.158,85.204,-104.095,167.912,47.739,158.869
C02446=1025.164,85.453,-104.113,167.915,47.735,158.869
C02447=1025.171,85.703,-104.131,167.918,47.731,158.868
C02448=1025.176,85.952,-104.149,167.920,47.728,158.868
C02449=1025.182,86.201,-104.167,167.923,47.724,158.867
C02450=1025.189,86.451,-104.185,167.925,47.719,158.867
C02451=1025.194,86.700,-104.203,167.928,47.716,158.866
C02452=1025.200,86.949,-104.221,167.931,47.712,158.866
C02453=1025.206,87.198,-104.239,167.934,47.708,158.866
C02454=1025.212,87.447,-104.257,167.936,47.704,158.865
C02455=1025.218,87.697,-104.276,167.939,47.701,158.865
C02456=1025.224,87.946,-104.294,167.941,47.696,158.864
C02457=1025.230,88.196,-104.312,167.944,47.692,158.864
C02458=1025.236,88.445,-104.330,167.947,47.689,158.864
C02459=1025.242,88.694,-104.348,167.949,47.685,158.863
C02460=1025.248,88.943,-104.367,167.951,47.680,158.863
C02461=1025.254,89.193,-104.385,167.954,47.677,158.862
C02462=1025.260,89.441,-104.403,167.957,47.673,158.862
C02463=1025.266,89.691,-104.421,167.960,47.669,158.862
C02464=1025.272,89.940,-104.440,167.961,47.666,158.861
C02465=1025.278,90.190,-104.458,167.964,47.662,158.861
C02466=1025.284,90.438,-104.476,167.967,47.658,158.861
C02467=1025.289,90.689,-104.495,167.970,47.654,158.860
C02468=1025.296,90.938,-104.513,167.972,47.651,158.860
C02469=1025.301,91.186,-104.532,167.975,47.647,158.859
C02470=1025.307,91.471,-104.553,167.977,47.642,158.859
C02471=1025.314,91.755,-104.574,167.981,47.638,158.858
C02472=1025.321,92.039,-104.595,167.984,47.634,158.858
C02473=1025.328,92.324,-104.616,167.986,47.629,158.858
C02474=1025.334,92.573,-104.634,167.989,47.625,158.857
C02475=1025.339,92.822,-104.653,167.992,47.622,158.857
C02476=1025.345,93.072,-104.671,167.995,47.618,158.856
C02477=1025.351,93.320,-104.690,167.997,47.614,158.856
C02478=1025.357,93.570,-104.709,167.999,47.611,158.856
C02479=1025.363,93.820,-104.727,168.002,47.606,158.855
C02480=1025.370,94.069,-104.745,168.005,47.602,158.855
C02481=1025.375,94.318,-104.764,168.008,47.599,158.854
C02482=1025.381,94.567,-104.782,168.010,47.595,158.854
C02483=1025.386,94.817,-104.802,168.012,47.591,158.854
C02484=1025.392,95.065,-104.820,168.015,47.587,158.853
C02485=1025.398,95.315,-104.838,168.018,47.584,158.853
C02486=1025.406,95.614,-104.861,168.021,47.579,158.852
C02487=1025.413,95.913,-104.883,168.024,47.574,158.852
C02488=1025.420,96.213,-104.905,168.027,47.570,158.851
C02489=1025.427,96.513,-104.928,168.030,47.565,158.851
C02490=1025.432,96.762,-104.946,168.033,47.561,158.851
C02491=1025.439,97.011,-104.965,168.036,47.558,158.850
C02492=1025.445,97.260,-104.984,168.038,47.553,158.850
C02493=1025.451,97.509,-105.003,168.041,47.550,158.849
C02494=1025.457,97.759,-105.020,168.043,47.546,158.849
C02495=1025.462,98.008,-105.039,168.046,47.542,158.849
C02496=1025.469,98.257,-105.058,168.049,47.538,158.848
C02497=1025.474,98.507,-105.077,168.052,47.534,158.848
C02498=1025.480,98.756,-105.095,168.053,47.530,158.847
C02499=1025.486,99.005,-105.113,168.056,47.526,158.847
C02500=1025.492,99.254,-105.133,168.059,47.523,158.847
C02501=1025.498,99.503,-105.151,168.062,47.519,158.846
C02502=1025.504,99.753,-105.171,168.065,47.515,158.846
C02503=1025.511,100.002,-105.189,168.067,47.512,158.845
C02504=1025.516,100.251,-105.208,168.070,47.508,158.845
C02505=1025.521,100.501,-105.227,168.072,47.504,158.845
C02506=1025.527,100.750,-105.245,168.075,47.500,158.844
C02507=1025.533,100.999,-105.265,168.078,47.496,158.844
C02508=1025.539,101.249,-105.284,168.080,47.493,158.843
C02509=1025.545,101.498,-105.302,168.083,47.489,158.843
C02510=1025.550,101.746,-105.321,168.086,47.485,158.843
C02511=1025.556,101.996,-105.341,168.088,47.481,158.842
C02512=1025.562,102.245,-105.359,168.090,47.477,158.842
C02513=1025.568,102.494,-105.378,168.093,47.474,158.841
C02514=1025.575,102.744,-105.397,168.096,47.470,158.841
C02515=1025.580,102.993,-105.416,168.099,47.466,158.841
C02516=1025.585,103.242,-105.435,168.102,47.462,158.840
C02517=1025.592,103.491,-105.454,168.103,47.459,158.840
C02518=1025.597,103.740,-105.473,168.106,47.455,158.840
C02519=1025.603,103.990,-105.492,168.109,47.451,158.839
C02520=1025.610,104.239,-105.511,168.112,47.447,158.839
C02521=1025.615,104.488,-105.530,168.115,47.444,158.838
C02522=1025.621,104.737,-105.550,168.117,47.440,158.838
C02523=1025.628,104.986,-105.569,168.120,47.436,158.838
C02524=1025.633,105.235,-105.588,168.123,47.433,158.837
C02525=1025.638,105.484,-105.607,168.125,47.429,158.837
C02526=1025.645,105.733,-105.626,168.128,47.424,158.836
C02527=1025.651,105.983,-105.645,168.130,47.421,158.836
C02528=1025.656,106.232,-105.664,168.133,47.417,158.836
C02529=1025.662,106.482,-105.683,168.136,47.413,158.835
C02530=1025.667,106.723,-105.701,168.138,47.410,158.835
C02531=1025.673,106.965,-105.720,168.141,47.406,158.835
C02532=1025.679,107.207,-105.739,168.143,47.402,158.834
C02533=1025.685,107.448,-105.758,168.146,47.398,158.834
C02534=1025.691,107.690,-105.776,168.149,47.395,158.833
C02535=1025.696,107.931,-105.794,168.151,47.391,158.833
C02536=1025.703,108.173,-105.813,168.154,47.387,158.833
C02537=1025.708,108.415,-105.831,168.156,47.384,158.832
C02538=1025.714,108.664,-105.850,168.159,47.380,158.832
C02539=1025.720,108.914,-105.870,168.162,47.376,158.831
C02540=1025.726,109.162,-105.889,168.164,47.373,158.831
C02541=1025.732,109.412,-105.908,168.167,47.369,158.831
C02542=1025.738,109.661,-105.927,168.170,47.365,158.830
C02543=1025.744,109.910,-105.946,168.172,47.361,158.830
C02544=1025.750,110.160,-105.965,168.175,47.357,158.829
C02545=1025.756,110.409,-105.985,168.178,47.353,158.829
C02546=1025.762,110.658,-106.005,168.180,47.350,158.829
C02547=1025.767,110.907,-106.024,168.183,47.346,158.828
C02548=1025.773,111.156,-106.043,168.186,47.342,158.828
C02549=1025.778,111.405,-106.063,168.189,47.338,158.827
C02550=1025.785,111.654,-106.081,168.191,47.335,158.827
C02551=1025.791,111.903,-106.101,168.194,47.331,158.827
C02552=1025.797,112.152,-106.121,168.196,47.327,158.826
C02553=1025.802,112.402,-106.140,168.199,47.324,158.826
C02554=1025.808,112.651,-106.160,168.202,47.320,158.826
C02555=1025.814,112.900,-106.179,168.205,47.316,158.825
C02556=1025.820,113.149,-106.198,168.208,47.312,158.825
C02557=1025.826,113.398,-106.218,168.210,47.309,158.824
C02558=1025.831,113.648,-106.237,168.212,47.305,158.824
C02559=1025.836,113.897,-106.258,168.215,47.301,158.824
C02560=1025.842,114.146,-106.277,168.218,47.297,158.823
C02561=1025.848,114.395,-106.297,168.221,47.294,158.823
C02562=1025.854,114.644,-106.316,168.223,47.291,158.823
C02563=1025.860,114.893,-106.336,168.226,47.287,158.822
C02564=1025.866,115.143,-106.356,168.229,47.283,158.822
C02565=1025.872,115.392,-106.376,168.232,47.280,158.822
C02566=1025.877,115.641,-106.395,168.235,47.276,158.821
C02567=1025.882,115.890,-106.415,168.237,47.272,158.821
C02568=1025.888,116.140,-106.435,168.239,47.269,158.820
C02569=1025.894,116.388,-106.455,168.242,47.265,158.820
C02570=1025.900,116.638,-106.474,168.245,47.261,158.820
C02571=1025.906,116.887,-106.494,168.248,47.257,158.819
C02572=1025.912,117.136,-106.513,168.250,47.254,158.819
C02573=1025.917,117.385,-106.534,168.253,47.250,158.818
C02574=1025.923,117.634,-106.554,168.256,47.246,158.818
C02575=1025.928,117.883,-106.573,168.259,47.243,158.818
C02576=1025.934,118.132,-106.593,168.261,47.239,158.817
C02577=1025.941,118.382,-106.612,168.263,47.235,158.817
C02578=1025.947,118.631,-106.632,168.266,47.232,158.817
C02579=1025.953,118.880,-106.652,168.269,47.228,158.816
C02580=1025.958,119.130,-106.672,168.272,47.224,158.816
C02581=1025.964,119.379,-106.692,168.275,47.220,158.815
C02582=1025.969,119.628,-106.711,168.278,47.217,158.815
C02583=1025.975,119.877,-106.731,168.281,47.214,158.815
C02584=1025.981,120.126,-106.751,168.283,47.210,158.814
C02585=1025.987,120.375,-106.770,168.286,47.206,158.814
C02586=1025.992,120.624,-106.791,168.289,47.203,158.814
C02587=1025.998,120.873,-106.811,168.291,47.199,158.813
C02588=1026.004,121.122,-106.830,168.294,47.195,158.813
C02589=1026.011,121.372,-106.851,168.297,47.191,158.813
C02590=1026.017,121.621,-106.870,168.300,47.188,158.812
C02591=1026.022,121.870,-106.890,168.302,47.184,158.812
C02592=1026.028,122.119,-106.910,168.305,47.180,158.811
C02593=1026.034,122.368,-106.930,168.308,47.177,158.811
C02594=1026.040,122.617,-106.950,168.311,47.173,158.811
C02595=1026.045,122.866,-106.969,168.313,47.169,158.810
C02596=1026.051,123.115,-106.989,168.316,47.165,158.810
C02597=1026.058,123.365,-107.010,168.319,47.162,158.810
C02598=1026.064,123.649,-107.033,168.322,47.157,158.809
C02599=1026.071,123.933,-107.055,168.325,47.153,158.809
C02600=1026.078,124.217,-107.078,168.328,47.149,158.808
C02601=1026.084,124.501,-107.101,168.331,47.144,158.808
C02602=1026.090,124.751,-107.121,168.334,47.141,158.807
C02603=1026.096,125.000,-107.141,168.337,47.137,158.807
C02604=1026.102,125.249,-107.160,168.340,47.133,158.807
C02605=1026.108,125.498,-107.180,168.342,47.129,158.806
C02606=1026.113,125.747,-107.201,168.345,47.126,158.806
C02607=1026.120,125.997,-107.221,168.348,47.122,158.805
C02608=1026.126,126.246,-107.241,168.351,47.118,158.805
C02609=1026.132,126.495,-107.261,168.354,47.114,158.805
C02610=1026.137,126.744,-107.280,168.357,47.111,158.804
C02611=1026.143,126.993,-107.301,168.360,47.107,158.804
C02612=1026.149,127.242,-107.321,168.363,47.103,158.804
C02613=1026.155,127.492,-107.341,168.365,47.100,158.803
C02614=1026.161,127.740,-107.361,168.367,47.096,158.803
C02615=1026.167,127.989,-107.381,168.370,47.092,158.802
C02616=1026.174,128.239,-107.401,168.373,47.089,158.802
C02617=1026.179,128.488,-107.421,168.376,47.085,158.802
C02618=1026.185,128.737,-107.441,168.379,47.081,158.801
C02619=1026.191,128.986,-107.461,168.382,47.077,158.801
C02620=1026.197,129.235,-107.482,168.384,47.073,158.800
C02621=1026.203,129.484,-107.502,168.387,47.069,158.800
C02622=1026.208,129.734,-107.521,168.390,47.066,158.800
C02623=1026.214,129.982,-107.541,168.393,47.062,158.799
C02624=1026.221,130.232,-107.562,168.396,47.058,158.799
C02625=1026.226,130.481,-107.582,168.399,47.054,158.799
C02626=1026.232,130.730,-107.602,168.402,47.051,158.798
C02627=1026.237,130.979,-107.623,168.405,47.048,158.798
C02628=1026.244,131.228,-107.644,168.407,47.044,158.797
C02629=1026.250,131.477,-107.664,168.410,47.040,158.797
C02630=1026.256,131.726,-107.684,168.413,47.037,158.797
C02631=1026.261,131.975,-107.705,168.416,47.033,158.796
C02632=1026.267,132.224,-107.725,168.418,47.029,158.796
C02633=1026.273,132.474,-107.746,168.421,47.025,158.796
C02634=1026.279,132.722,-107.766,168.424,47.022,158.795
C02635=1026.285,132.972,-107.787,168.427,47.018,158.795
C02636=1026.291,133.221,-107.807,168.430,47.015,158.795
C02637=1026.296,133.470,-107.828,168.433,47.011,158.794
C02638=1026.302,133.718,-107.848,168.436,47.008,158.794
C02639=1026.308,133.968,-107.869,168.438,47.004,158.793
C02640=1026.314,134.217,-107.889,168.441,47.000,158.793
C02641=1026.319,134.466,-107.909,168.444,46.997,158.793
C02642=1026.326,134.716,-107.930,168.447,46.993,158.792
C02643=1026.331,134.964,-107.951,168.450,46.989,158.792
C02644=1026.337,135.213,-107.971,168.453,46.985,158.792
C02645=1026.343,135.463,-107.992,168.455,46.982,158.791
C02646=1026.349,135.712,-108.012,168.458,46.978,158.791
C02647=1026.355,135.960,-108.033,168.461,46.975,158.791
C02648=1026.361,136.210,-108.054,168.464,46.971,158.790
C02649=1026.367,136.459,-108.074,168.467,46.968,158.790
C02650=1026.372,136.708,-108.094,168.470,46.964,158.790
C02651=1026.378,136.957,-108.116,168.473,46.960,158.789
C02652=1026.384,137.206,-108.136,168.476,46.956,158.789
C02653=1026.389,137.455,-108.157,168.479,46.953,158.788
C02654=1026.396,137.705,-108.177,168.482,46.949,158.788
C02655=1026.401,137.953,-108.198,168.485,46.945,158.788
C02656=1026.407,138.203,-108.219,168.488,46.942,158.787
C02657=1026.413,138.452,-108.239,168.491,46.938,158.787
C02658=1026.419,138.700,-108.260,168.493,46.935,158.787
C02659=1026.425,138.950,-108.281,168.496,46.931,158.786
C02660=1026.430,139.199,-108.302,168.498,46.928,158.786
C02661=1026.437,139.448,-108.323,168.501,46.924,158.786
C02662=1026.443,139.731,-108.346,168.505,46.920,158.785
C02663=1026.449,140.016,-108.370,168.508,46.916,158.785
C02664=1026.456,140.300,-108.394,168.512,46.912,158.784
C02665=1026.462,140.584,-108.418,168.515,46.908,158.784
C02666=1026.469,140.833,-108.439,168.518,46.904,158.784
C02667=1026.474,141.082,-108.460,168.521,46.900,158.783
C02668=1026.480,141.332,-108.480,168.524,46.897,158.783
C02669=1026.486,141.581,-108.502,168.527,46.894,158.783
C02670=1026.491,141.830,-108.523,168.530,46.890,158.782
C02671=1026.498,142.079,-108.544,168.532,46.886,158.782
C02672=1026.503,142.328,-108.564,168.535,46.883,158.782
C02673=1026.509,142.577,-108.586,168.539,46.880,158.781
C02674=1026.515,142.826,-108.606,168.541,46.876,158.781
C02675=1026.520,143.075,-108.628,168.544,46.872,158.781
C02676=1026.527,143.324,-108.649,168.547,46.868,158.780
C02677=1026.532,143.573,-108.669,168.550,46.865,158.780
C02678=1026.538,143.822,-108.691,168.553,46.861,158.779
C02679=1026.544,144.071,-108.712,168.556,46.858,158.779
C02680=1026.550,144.320,-108.733,168.559,46.854,158.779
C02681=1026.556,144.569,-108.753,168.562,46.851,158.778
C02682=1026.562,144.818,-108.775,168.565,46.847,158.778
C02683=1026.567,145.067,-108.795,168.568,46.843,158.778
C02684=1026.573,145.317,-108.817,168.571,46.839,158.777
C02685=1026.579,145.565,-108.838,168.574,46.836,158.777
C02686=1026.586,145.815,-108.859,168.577,46.833,158.777
C02687=1026.591,146.063,-108.880,168.580,46.829,158.776
C02688=1026.597,146.312,-108.901,168.583,46.825,158.776
C02689=1026.603,146.562,-108.922,168.586,46.822,158.776
C02690=1026.609,146.811,-108.944,168.589,46.819,158.775
C02691=1026.614,147.059,-108.965,168.592,46.815,158.775
C02692=1026.620,147.309,-108.986,168.595,46.811,158.775
C02693=1026.626,147.558,-109.007,168.598,46.808,158.774
C02694=1026.632,147.807,-109.029,168.601,46.804,158.774
C02695=1026.637,148.055,-109.050,168.604,46.801,158.774
C02696=1026.643,148.305,-109.071,168.607,46.797,158.773
C02697=1026.649,148.554,-109.092,168.610,46.794,158.773
C02698=1026.655,148.803,-109.114,168.613,46.790,158.773
C02699=1026.661,149.051,-109.135,168.616,46.787,158.772
C02700=1026.667,149.301,-109.157,168.618,46.783,158.772
C02701=1026.672,149.550,-109.177,168.622,46.780,158.772
C02702=1026.678,149.799,-109.199,168.625,46.776,158.771
C02703=1026.684,150.048,-109.221,168.628,46.773,158.771
C02704=1026.689,150.297,-109.242,168.631,46.770,158.771
C02705=1026.695,150.546,-109.264,168.634,46.766,158.770
C02706=1026.701,150.795,-109.285,168.637,46.762,158.770
C02707=1026.707,151.044,-109.306,168.639,46.758,158.770
C02708=1026.712,151.293,-109.327,168.643,46.755,158.769
C02709=1026.718,151.542,-109.349,168.646,46.752,158.769
C02710=1026.725,151.791,-109.371,168.648,46.748,158.769
C02711=1026.730,152.040,-109.392,168.652,46.745,158.768
C02712=1026.736,152.289,-109.414,168.655,46.741,158.768
C02713=1026.742,152.538,-109.435,168.658,46.738,158.768
C02714=1026.748,152.787,-109.457,168.660,46.734,158.767
C02715=1026.753,153.036,-109.479,168.664,46.731,158.767
C02716=1026.759,153.285,-109.500,168.667,46.727,158.767
C02717=1026.765,153.534,-109.522,168.669,46.724,158.766
C02718=1026.771,153.782,-109.543,168.674,46.720,158.766
C02719=1026.777,154.032,-109.565,168.677,46.717,158.766
C02720=1026.783,154.281,-109.586,168.680,46.713,158.765
C02721=1026.788,154.530,-109.608,168.683,46.710,158.765
C02722=1026.794,154.779,-109.630,168.686,46.706,158.765
C02723=1026.800,155.028,-109.651,168.689,46.703,158.764
C02724=1026.806,155.277,-109.673,168.692,46.700,158.764
C02725=1026.811,155.526,-109.695,168.695,46.696,158.764
C02726=1026.818,155.810,-109.719,168.698,46.692,158.763
C02727=1026.824,156.094,-109.744,168.702,46.688,158.763
C02728=1026.831,156.377,-109.769,168.705,46.684,158.763
C02729=1026.838,156.661,-109.793,168.708,46.680,158.762
C02730=1026.844,156.910,-109.816,168.711,46.677,158.762
C02731=1026.850,157.160,-109.838,168.715,46.673,158.762
C02732=1026.855,157.408,-109.859,168.718,46.670,158.762
C02733=1026.862,157.657,-109.880,168.721,46.666,158.761
C02734=1026.867,157.907,-109.903,168.724,46.663,158.761
C02735=1026.873,158.155,-109.924,168.727,46.660,158.761
C02736=1026.879,158.404,-109.946,168.730,46.656,158.760
C02737=1026.885,158.653,-109.968,168.733,46.652,158.760
C02738=1026.890,158.902,-109.990,168.737,46.649,158.760
C02739=1026.896,159.151,-110.011,168.739,46.646,158.759
C02740=1026.902,159.400,-110.033,168.742,46.642,158.759
C02741=1026.908,159.650,-110.055,168.746,46.639,158.759
C02742=1026.913,159.898,-110.078,168.749,46.636,158.758
C02743=1026.919,160.147,-110.099,168.752,46.632,158.758
C02744=1026.925,160.396,-110.122,168.755,46.629,158.758
C02745=1026.930,160.645,-110.144,168.758,46.626,158.757
C02746=1026.936,160.894,-110.166,168.761,46.623,158.757
C02747=1026.942,161.143,-110.189,168.765,46.619,158.757
C02748=1026.946,161.392,-110.211,168.768,46.616,158.757
C02749=1026.953,161.640,-110.233,168.771,46.613,158.756
C02750=1026.958,161.890,-110.255,168.774,46.609,158.756
C02751=1026.964,162.139,-110.278,168.778,46.606,158.756
C02752=1026.969,162.388,-110.300,168.780,46.602,158.755
C02753=1026.975,162.637,-110.322,168.784,46.599,158.755
C02754=1026.981,162.886,-110.345,168.787,46.596,158.755
C02755=1026.986,163.135,-110.367,168.790,46.593,158.755
C02756=1026.992,163.383,-110.389,168.793,46.590,158.754
C02757=1026.997,163.633,-110.411,168.796,46.586,158.754
C02758=1027.003,163.882,-110.434,168.799,46.583,158.754
C02759=1027.009,164.130,-110.455,168.802,46.579,158.753
C02760=1027.014,164.379,-110.478,168.805,46.576,158.753
C02761=1027.020,164.628,-110.501,168.808,46.573,158.753
C02762=1027.026,164.877,-110.523,168.811,46.570,158.753
C02763=1027.032,165.126,-110.546,168.816,46.566,158.752
C02764=1027.037,165.375,-110.568,168.819,46.563,158.752
C02765=1027.043,165.624,-110.591,168.822,46.560,158.752
C02766=1027.049,165.873,-110.612,168.825,46.557,158.752
C02767=1027.055,166.122,-110.635,168.828,46.553,158.751
C02768=1027.060,166.371,-110.657,168.831,46.550,158.751
C02769=1027.065,166.619,-110.680,168.834,46.546,158.751
C02770=1027.072,166.868,-110.702,168.837,46.543,158.750
C02771=1027.077,167.118,-110.725,168.840,46.540,158.750
C02772=1027.083,167.366,-110.748,168.844,46.536,158.750
C02773=1027.089,167.615,-110.770,168.848,46.534,158.750
C02774=1027.094,167.864,-110.792,168.851,46.530,158.749
C02775=1027.100,168.113,-110.815,168.854,46.527,158.749
C02776=1027.105,168.362,-110.838,168.857,46.523,158.749
C02777=1027.112,168.611,-110.859,168.860,46.520,158.748
C02778=1027.117,168.860,-110.882,168.863,46.517,158.748
C02779=1027.123,169.109,-110.905,168.867,46.513,158.748
C02780=1027.129,169.358,-110.927,168.870,46.510,158.748
C02781=1027.135,169.607,-110.950,168.873,46.507,158.747
C02782=1027.140,169.855,-110.972,168.876,46.504,158.747
C02783=1027.146,170.104,-110.995,168.880,46.501,158.747
C02784=1027.152,170.353,-111.017,168.883,46.497,158.746
C02785=1027.158,170.602,-111.040,168.887,46.494,158.746
C02786=1027.163,170.851,-111.063,168.890,46.490,158.746
C02787=1027.169,171.100,-111.085,168.893,46.487,158.746
C02788=1027.175,171.349,-111.107,168.896,46.483,158.745
C02789=1027.181,171.598,-111.130,168.899,46.480,158.745
C02790=1027.188,171.881,-111.156,168.903,46.477,158.745
C02791=1027.194,172.165,-111.182,168.907,46.473,158.744
C02792=1027.201,172.448,-111.208,168.911,46.469,158.744
C02793=1027.207,172.732,-111.233,168.915,46.466,158.744
C02794=1027.214,172.981,-111.256,168.918,46.462,158.744
C02795=1027.220,173.230,-111.279,168.921,46.459,158.743
C02796=1027.225,173.479,-111.302,168.924,46.455,158.743
C02797=1027.230,173.727,-111.324,168.927,46.452,158.743
C02798=1027.237,173.975,-111.347,168.932,46.449,158.743
C02799=1027.243,174.224,-111.370,168.935,46.445,158.742
C02800=1027.248,174.474,-111.392,168.938,46.442,158.742
C02801=1027.254,174.723,-111.415,168.941,46.439,158.742
C02802=1027.261,174.972,-111.437,168.945,46.436,158.741
C02803=1027.267,175.221,-111.460,168.948,46.433,158.741
C02804=1027.272,175.470,-111.483,168.951,46.429,158.741
C02805=1027.278,175.719,-111.506,168.954,46.426,158.741
C02806=1027.285,175.967,-111.529,168.958,46.422,158.740
C02807=1027.290,176.216,-111.552,168.962,46.419,158.740
C02808=1027.296,176.465,-111.575,168.965,46.416,158.740
C02809=1027.302,176.714,-111.597,168.968,46.412,158.739
C02810=1027.308,176.963,-111.620,168.972,46.409,158.739
C02811=1027.314,177.211,-111.643,168.975,46.406,158.739
C02812=1027.320,177.460,-111.666,168.978,46.403,158.739
C02813=1027.325,177.709,-111.689,168.982,46.399,158.738
C02814=1027.332,177.958,-111.711,168.985,46.396,158.738
C02815=1027.338,178.207,-111.734,168.988,46.393,158.738
C02816=1027.343,178.456,-111.757,168.993,46.389,158.738
C02817=1027.350,178.705,-111.780,168.996,46.386,158.737
C02818=1027.355,178.954,-111.803,168.999,46.383,158.737
C02819=1027.362,179.203,-111.825,169.002,46.380,158.737
C02820=1027.368,179.452,-111.848,169.006,46.376,158.736
C02821=1027.373,179.701,-111.871,169.009,46.373,158.736
C02822=1027.379,179.949,-111.894,169.012,46.369,158.736
C02823=1027.386,180.198,-111.917,169.016,46.366,158.736
C02824=1027.391,180.447,-111.940,169.020,46.363,158.735
C02825=1027.398,180.697,-111.963,169.023,46.360,158.735
C02826=1027.404,180.945,-111.987,169.027,46.356,158.735
C02827=1027.409,181.194,-112.010,169.030,46.353,158.735
C02828=1027.416,181.442,-112.032,169.033,46.350,158.734
C02829=1027.422,181.691,-112.055,169.037,46.347,158.734
C02830=1027.428,181.941,-112.078,169.040,46.344,158.734
C02831=1027.434,182.190,-112.101,169.044,46.340,158.734
C02832=1027.440,182.438,-112.124,169.048,46.337,158.733
C02833=1027.446,182.687,-112.147,169.051,46.334,158.733
C02834=1027.451,182.936,-112.171,169.055,46.330,158.733
C02835=1027.457,183.185,-112.194,169.058,46.327,158.733
C02836=1027.464,183.434,-112.218,169.061,46.324,158.732
C02837=1027.469,183.683,-112.241,169.064,46.321,158.732
C02838=1027.475,183.931,-112.265,169.069,46.318,158.732
C02839=1027.480,184.180,-112.288,169.072,46.315,158.732
C02840=1027.486,184.429,-112.312,169.075,46.312,158.731
C02841=1027.492,184.678,-112.335,169.078,46.309,158.731
C02842=1027.497,184.927,-112.360,169.083,46.306,158.731
C02843=1027.503,185.176,-112.383,169.086,46.303,158.731
C02844=1027.508,185.424,-112.407,169.089,46.300,158.731
C02845=1027.514,185.673,-112.430,169.093,46.296,158.730
C02846=1027.520,185.921,-112.453,169.096,46.293,158.730
C02847=1027.526,186.171,-112.477,169.100,46.291,158.730
C02848=1027.532,186.420,-112.501,169.103,46.288,158.730
C02849=1027.537,186.669,-112.525,169.107,46.284,158.730
C02850=1027.543,186.917,-112.548,169.110,46.281,158.729
C02851=1027.548,187.166,-112.571,169.114,46.278,158.729
C02852=1027.554,187.415,-112.596,169.118,46.275,158.729
C02853=1027.560,187.664,-112.619,169.121,46.272,158.729
C02854=1027.566,187.947,-112.646,169.125,46.269,158.729
C02855=1027.573,188.229,-112.673,169.129,46.265,158.728
C02856=1027.580,188.513,-112.700,169.134,46.262,158.728
C02857=1027.587,188.795,-112.727,169.137,46.258,158.728
C02858=1027.592,189.045,-112.751,169.141,46.255,158.728
C02859=1027.598,189.293,-112.774,169.144,46.252,158.727
C02860=1027.604,189.542,-112.798,169.148,46.249,158.727
C02861=1027.609,189.791,-112.822,169.151,46.246,158.727
C02862=1027.615,190.039,-112.846,169.155,46.243,158.727
C02863=1027.621,190.288,-112.870,169.159,46.240,158.726
C02864=1027.627,190.537,-112.894,169.162,46.237,158.726
C02865=1027.632,190.786,-112.917,169.166,46.234,158.726
C02866=1027.638,191.034,-112.941,169.170,46.231,158.726
C02867=1027.645,191.283,-112.965,169.173,46.228,158.726
C02868=1027.650,191.532,-112.989,169.177,46.225,158.726
C02869=1027.656,191.781,-113.012,169.181,46.222,158.725
C02870=1027.662,192.030,-113.037,169.185,46.219,158.725
C02871=1027.668,192.278,-113.061,169.188,46.216,158.725
C02872=1027.674,192.527,-113.084,169.191,46.213,158.725
C02873=1027.680,192.776,-113.109,169.195,46.210,158.725
C02874=1027.686,193.025,-113.132,169.199,46.207,158.724
C02875=1027.692,193.274,-113.157,169.203,46.204,158.724
C02876=1027.698,193.523,-113.180,169.206,46.201,158.724
C02877=1027.703,193.771,-113.204,169.209,46.198,158.724
C02878=1027.710,194.020,-113.228,169.214,46.195,158.724
C02879=1027.716,194.268,-113.252,169.217,46.192,158.723
C02880=1027.721,194.518,-113.276,169.221,46.189,158.723
C02881=1027.727,194.767,-113.300,169.224,46.186,158.723
C02882=1027.733,195.015,-113.324,169.229,46.182,158.723
C02883=1027.739,195.264,-113.348,169.232,46.179,158.723
C02884=1027.744,195.513,-113.372,169.236,46.176,158.722
C02885=1027.751,195.762,-113.396,169.239,46.173,158.722
C02886=1027.756,196.010,-113.421,169.244,46.171,158.722
C02887=1027.763,196.259,-113.445,169.247,46.168,158.722
C02888=1027.769,196.508,-113.468,169.251,46.165,158.722
C02889=1027.775,196.757,-113.493,169.254,46.162,158.721
C02890=1027.781,197.005,-113.516,169.258,46.159,158.721
C02891=1027.787,197.254,-113.541,169.262,46.156,158.721
C02892=1027.793,197.503,-113.565,169.265,46.153,158.721
C02893=1027.799,197.752,-113.589,169.269,46.149,158.721
C02894=1027.805,198.000,-113.613,169.273,46.146,158.720
C02895=1027.811,198.250,-113.638,169.277,46.143,158.720
C02896=1027.817,198.498,-113.661,169.281,46.141,158.720
C02897=1027.823,198.747,-113.686,169.285,46.138,158.720
C02898=1027.829,198.995,-113.710,169.289,46.135,158.720
C02899=1027.835,199.244,-113.734,169.292,46.132,158.720
C02900=1027.841,199.493,-113.758,169.296,46.128,158.719
C02901=1027.847,199.742,-113.782,169.300,46.126,158.719
C02902=1027.853,199.990,-113.807,169.304,46.122,158.719
C02903=1027.860,200.239,-113.831,169.307,46.119,158.719
C02904=1027.865,200.488,-113.856,169.312,46.117,158.719
C02905=1027.871,200.737,-113.880,169.315,46.114,158.719
C02906=1027.877,200.986,-113.904,169.319,46.111,158.718
C02907=1027.882,201.234,-113.929,169.323,46.108,158.718
C02908=1027.889,201.483,-113.953,169.327,46.105,158.718
C02909=1027.894,201.732,-113.978,169.330,46.102,158.718
C02910=1027.900,201.980,-114.003,169.335,46.100,158.718
C02911=1027.906,202.229,-114.027,169.338,46.097,158.718
C02912=1027.912,202.478,-114.052,169.342,46.094,158.717
C02913=1027.918,202.727,-114.077,169.346,46.091,158.717
C02914=1027.924,202.975,-114.101,169.350,46.088,158.717
C02915=1027.930,203.224,-114.126,169.353,46.085,158.717
C02916=1027.935,203.472,-114.150,169.358,46.083,158.717
C02917=1027.941,203.722,-114.175,169.361,46.080,158.717
C02918=1027.966,204.765,-114.279,169.737,46.183,158.781
C02919=1027.977,205.147,-114.319,169.742,46.180,158.781
C02920=1027.987,205.530,-114.359,169.746,46.176,158.781
C02921=1027.998,205.912,-114.399,169.750,46.173,158.781
C02922=1028.008,206.294,-114.439,169.755,46.170,158.780
C02923=1028.015,206.542,-114.465,169.757,46.169,158.781
C02924=1028.021,206.791,-114.492,169.761,46.166,158.780
C02925=1028.027,207.040,-114.518,169.763,46.164,158.780
C02926=1028.034,207.289,-114.544,169.766,46.162,158.780
C02927=1028.041,207.537,-114.570,169.769,46.160,158.780
C02928=1028.048,207.786,-114.596,169.772,46.158,158.780
C02929=1028.054,208.034,-114.622,169.775,46.157,158.780
C02930=1028.061,208.283,-114.649,169.778,46.154,158.780
C02931=1028.067,208.531,-114.676,169.781,46.152,158.780
C02932=1028.074,208.780,-114.702,169.784,46.150,158.780
C02933=1028.081,209.028,-114.728,169.786,46.148,158.779
C02934=1028.087,209.277,-114.755,169.789,46.147,158.779
C02935=1028.093,209.525,-114.780,169.793,46.144,158.779
C02936=1028.101,209.774,-114.807,169.795,46.142,158.779
C02937=1028.107,210.022,-114.833,169.798,46.140,158.779
C02938=1028.113,210.271,-114.860,169.801,46.139,158.779
C02939=1028.120,210.519,-114.886,169.804,46.137,158.779
C02940=1028.127,210.768,-114.912,169.806,46.135,158.779
C02941=1028.133,211.016,-114.939,169.810,46.132,158.779
C02942=1028.140,211.265,-114.965,169.813,46.131,158.779
C02943=1028.147,211.513,-114.992,169.815,46.129,158.779
C02944=1028.153,211.762,-115.019,169.819,46.127,158.779
C02945=1028.160,212.010,-115.046,169.821,46.125,158.779
C02946=1028.166,212.259,-115.072,169.824,46.123,158.778
C02947=1028.173,212.508,-115.099,169.827,46.121,158.778
C02948=1028.179,212.756,-115.125,169.830,46.119,158.778
C02949=1028.186,213.005,-115.152,169.833,46.117,158.778
C02950=1028.193,213.253,-115.178,169.836,46.115,158.778
C02951=1028.199,213.502,-115.205,169.839,46.114,158.778
C02952=1028.206,213.750,-115.232,169.842,46.111,158.778
C02953=1028.212,213.998,-115.259,169.845,46.110,158.778
C02954=1028.219,214.247,-115.285,169.848,46.108,158.778
C02955=1028.225,214.495,-115.312,169.851,46.106,158.778
C02956=1028.232,214.744,-115.338,169.854,46.104,158.778
C02957=1028.239,214.993,-115.364,169.856,46.102,158.778
C02958=1028.245,215.241,-115.392,169.860,46.100,158.778
C02959=1028.252,215.489,-115.418,169.863,46.099,158.778
C02960=1028.258,215.738,-115.445,169.865,46.097,158.778
C02961=1028.265,215.986,-115.471,169.869,46.095,158.778
C02962=1028.272,216.235,-115.499,169.871,46.093,158.777
C02963=1028.279,216.483,-115.525,169.875,46.091,158.777
C02964=1028.285,216.732,-115.552,169.878,46.089,158.777
C02965=1028.292,216.981,-115.579,169.880,46.087,158.777
C02966=1028.299,217.228,-115.605,169.884,46.086,158.777
C02967=1028.305,217.477,-115.632,169.886,46.084,158.777
C02968=1028.312,217.726,-115.659,169.890,46.081,158.777
C02969=1028.318,217.974,-115.685,169.893,46.080,158.777
C02970=1028.326,218.222,-115.713,169.895,46.078,158.777
C02971=1028.332,218.472,-115.740,169.899,46.076,158.777
C02972=1028.338,218.720,-115.766,169.901,46.074,158.777
C02973=1028.345,218.968,-115.793,169.905,46.073,158.777
C02974=1028.352,219.217,-115.820,169.908,46.071,158.777
C02975=1028.362,219.604,-115.862,169.912,46.068,158.777
C02976=1028.372,219.991,-115.904,169.918,46.065,158.777
C02977=1028.382,220.378,-115.946,169.922,46.062,158.777
C02978=1028.393,220.766,-115.988,169.926,46.060,158.777
C02979=1028.399,221.014,-116.016,169.929,46.058,158.777
C02980=1028.406,221.263,-116.043,169.933,46.056,158.777
C02981=1028.412,221.511,-116.070,169.935,46.055,158.777
C02982=1028.419,221.759,-116.096,169.939,46.053,158.777
C02983=1028.426,222.008,-116.124,169.942,46.051,158.776
C02984=1028.432,222.256,-116.152,169.944,46.050,158.776
C02985=1028.439,222.505,-116.179,169.948,46.047,158.776
C02986=1028.445,222.753,-116.206,169.951,46.046,158.776
C02987=1028.452,223.002,-116.233,169.954,46.044,158.776
C02988=1028.459,223.250,-116.260,169.957,46.042,158.776
C02989=1028.465,223.499,-116.287,169.960,46.041,158.776
C02990=1028.472,223.747,-116.314,169.963,46.039,158.776
C02991=1028.478,223.995,-116.342,169.966,46.037,158.776
C02992=1028.485,224.244,-116.369,169.970,46.036,158.776
C02993=1028.492,224.492,-116.396,169.972,46.034,158.776
C02994=1028.498,224.740,-116.423,169.975,46.032,158.776
C02995=1028.505,224.989,-116.450,169.979,46.031,158.776
C02996=1028.511,225.238,-116.478,169.981,46.029,158.776
C02997=1028.518,225.486,-116.504,169.985,46.027,158.776
C02998=1028.525,225.735,-116.532,169.987,46.025,158.776
C02999=1028.532,225.983,-116.560,169.991,46.023,158.776
C03000=1028.538,226.231,-116.587,169.994,46.022,158.776
C03001=1028.545,226.480,-116.614,169.996,46.020,158.776
C03002=1028.552,226.728,-116.641,170.000,46.018,158.776
C03003=1028.558,226.977,-116.669,170.003,46.017,158.776
C03004=1028.565,227.226,-116.696,170.006,46.015,158.776
C03005=1028.572,227.474,-116.723,170.009,46.013,158.776
C03006=1028.578,227.721,-116.751,170.013,46.012,158.776
C03007=1028.585,227.970,-116.778,170.016,46.010,158.776
C03008=1028.592,228.218,-116.806,170.018,46.009,158.776
C03009=1028.598,228.467,-116.834,170.022,46.007,158.776
C03010=1028.605,228.716,-116.861,170.025,46.005,158.776
C03011=1028.611,228.964,-116.889,170.028,46.004,158.776
C03012=1028.617,229.212,-116.916,170.031,46.002,158.776
C03013=1028.624,229.460,-116.944,170.035,46.001,158.776
C03014=1028.631,229.709,-116.971,170.037,45.999,158.776
C03015=1028.637,229.957,-116.999,170.040,45.997,158.776
C03016=1028.644,230.206,-117.027,170.044,45.996,158.776
C03017=1028.651,230.454,-117.055,170.047,45.994,158.776
C03018=1028.657,230.703,-117.082,170.051,45.993,158.776
C03019=1028.664,230.951,-117.110,170.053,45.990,158.776
C03020=1028.670,231.199,-117.137,170.057,45.989,158.776
C03021=1028.677,231.447,-117.165,170.060,45.987,158.776
C03022=1028.683,231.696,-117.194,170.062,45.986,158.776
C03023=1028.690,231.944,-117.221,170.066,45.984,158.776
C03024=1028.696,232.193,-117.249,170.069,45.983,158.776
C03025=1028.703,232.441,-117.277,170.073,45.981,158.776
C03026=1028.710,232.690,-117.304,170.075,45.980,158.776
C03027=1028.716,232.938,-117.332,170.079,45.978,158.776
C03028=1028.723,233.187,-117.360,170.082,45.977,158.776
C03029=1028.729,233.435,-117.388,170.085,45.976,158.776
C03030=1028.735,233.683,-117.416,170.088,45.974,158.777
C03031=1028.746,234.062,-117.458,170.093,45.972,158.776
C03032=1028.756,234.442,-117.501,170.097,45.969,158.776
C03033=1028.766,234.822,-117.544,170.103,45.967,158.777
C03034=1028.776,235.202,-117.587,170.108,45.964,158.777
C03035=1028.783,235.450,-117.614,170.111,45.963,158.777
C03036=1028.789,235.699,-117.642,170.114,45.961,158.777
C03037=1028.796,235.946,-117.670,170.117,45.960,158.777
C03038=1028.803,236.195,-117.698,170.121,45.958,158.777
C03039=1028.809,236.444,-117.727,170.124,45.957,158.777
C03040=1028.815,236.692,-117.754,170.127,45.956,158.777
C03041=1028.822,236.941,-117.782,170.130,45.954,158.777
C03042=1028.829,237.188,-117.810,170.134,45.953,158.777
C03043=1028.836,237.437,-117.838,170.137,45.951,158.777
C03044=1028.843,237.685,-117.866,170.140,45.950,158.777
C03045=1028.849,237.933,-117.895,170.143,45.948,158.777
C03046=1028.855,238.182,-117.923,170.147,45.947,158.777
C03047=1028.862,238.430,-117.950,170.150,45.945,158.777
C03048=1028.869,238.678,-117.979,170.153,45.944,158.777
C03049=1028.875,238.927,-118.007,170.156,45.942,158.777
C03050=1028.882,239.175,-118.035,170.160,45.941,158.777
C03051=1028.889,239.423,-118.063,170.163,45.939,158.777
C03052=1028.895,239.672,-118.091,170.167,45.938,158.778
C03053=1028.902,239.920,-118.119,170.170,45.937,158.778
C03054=1028.908,240.168,-118.148,170.173,45.935,158.778
C03055=1028.915,240.417,-118.176,170.176,45.934,158.778
C03056=1028.921,240.665,-118.205,170.180,45.932,158.778
C03057=1028.928,240.913,-118.232,170.183,45.931,158.778
C03058=1028.934,241.161,-118.261,170.186,45.929,158.778
C03059=1028.941,241.410,-118.289,170.189,45.928,158.778
C03060=1028.948,241.659,-118.319,170.192,45.927,158.778
C03061=1028.954,241.907,-118.346,170.196,45.925,158.778
C03062=1028.961,242.155,-118.375,170.199,45.924,158.778
C03063=1028.968,242.403,-118.404,170.203,45.923,158.778
C03064=1028.974,242.652,-118.432,170.206,45.922,158.778
C03065=1028.981,242.899,-118.461,170.209,45.920,158.778
C03066=1028.987,243.148,-118.489,170.212,45.919,158.778
C03067=1028.994,243.396,-118.517,170.216,45.917,158.778
C03068=1029.000,243.644,-118.546,170.219,45.916,158.779
C03069=1029.007,243.893,-118.574,170.223,45.915,158.779
C03070=1029.014,244.141,-118.603,170.225,45.913,158.779
C03071=1029.020,244.390,-118.631,170.229,45.912,158.779
C03072=1029.026,244.638,-118.660,170.232,45.911,158.779
C03073=1029.032,244.886,-118.689,170.236,45.909,158.779
C03074=1029.039,245.134,-118.718,170.239,45.909,158.779
C03075=1029.046,245.382,-118.747,170.243,45.907,158.779
C03076=1029.052,245.631,-118.775,170.246,45.906,158.779
C03077=1029.058,245.879,-118.804,170.250,45.905,158.780
C03078=1029.065,246.128,-118.833,170.252,45.903,158.780
C03079=1029.072,246.376,-118.862,170.256,45.902,158.780
C03080=1029.078,246.624,-118.891,170.259,45.901,158.780
C03081=1029.084,246.873,-118.919,170.263,45.899,158.780
C03082=1029.091,247.120,-118.948,170.266,45.899,158.780
C03083=1029.097,247.368,-118.977,170.270,45.897,158.780
C03084=1029.104,247.617,-119.006,170.273,45.896,158.780
C03085=1029.110,247.865,-119.035,170.277,45.895,158.780
C03086=1029.117,248.114,-119.064,170.280,45.894,158.781
C03087=1029.127,248.487,-119.108,170.285,45.892,158.781
C03088=1029.136,248.861,-119.151,170.290,45.890,158.781
C03089=1029.146,249.234,-119.194,170.295,45.888,158.781
C03090=1029.156,249.608,-119.238,170.300,45.886,158.781
C03091=1029.162,249.856,-119.267,170.304,45.885,158.781
C03092=1029.169,250.104,-119.296,170.307,45.884,158.781
C03093=1029.176,250.352,-119.325,170.311,45.883,158.782
C03094=1029.182,250.601,-119.354,170.314,45.881,158.782
C03095=1029.189,250.849,-119.383,170.317,45.881,158.782
C03096=1029.196,251.097,-119.412,170.321,45.879,158.782
C03097=1029.203,251.346,-119.441,170.324,45.878,158.782
C03098=1029.209,251.594,-119.470,170.328,45.877,158.782
C03099=1029.215,251.842,-119.499,170.331,45.876,158.782
C03100=1029.221,252.090,-119.528,170.335,45.874,158.782
C03101=1029.229,252.338,-119.557,170.338,45.874,158.783
C03102=1029.235,252.587,-119.586,170.342,45.872,158.783
C03103=1029.242,252.834,-119.616,170.346,45.871,158.783
C03104=1029.249,253.083,-119.645,170.348,45.870,158.783
C03105=1029.255,253.331,-119.674,170.352,45.869,158.783
C03106=1029.262,253.579,-119.703,170.355,45.867,158.783
C03107=1029.269,253.828,-119.732,170.359,45.866,158.783
C03108=1029.275,254.076,-119.761,170.362,45.865,158.783
C03109=1029.281,254.324,-119.790,170.366,45.864,158.784
C03110=1029.289,254.572,-119.820,170.370,45.863,158.784
C03111=1029.295,254.820,-119.849,170.373,45.862,158.784
C03112=1029.302,255.069,-119.878,170.377,45.861,158.784
C03113=1029.308,255.317,-119.907,170.380,45.859,158.784
C03114=1029.315,255.565,-119.936,170.384,45.858,158.784
C03115=1029.322,255.813,-119.966,170.387,45.857,158.784
C03116=1029.329,256.061,-119.995,170.390,45.856,158.785
C03117=1029.336,256.310,-120.024,170.395,45.855,158.785
C03118=1029.342,256.558,-120.053,170.397,45.854,158.785
C03119=1029.348,256.806,-120.083,170.401,45.853,158.785
C03120=1029.356,257.054,-120.112,170.405,45.852,158.785
C03121=1029.362,257.302,-120.141,170.408,45.850,158.785
C03122=1029.369,257.550,-120.171,170.412,45.849,158.786
C03123=1029.376,257.799,-120.200,170.416,45.848,158.786
C03124=1029.382,258.047,-120.229,170.419,45.847,158.786
C03125=1029.389,258.295,-120.259,170.423,45.846,158.786
C03126=1029.397,258.543,-120.288,170.426,45.845,158.786
C03127=1029.403,258.792,-120.317,170.430,45.844,158.786
C03128=1029.410,259.040,-120.347,170.434,45.843,158.787
C03129=1029.416,259.288,-120.376,170.437,45.841,158.787
C03130=1029.423,259.537,-120.406,170.441,45.841,158.787
C03131=1029.430,259.784,-120.435,170.445,45.840,158.787
C03132=1029.437,260.033,-120.464,170.447,45.838,158.787
C03133=1029.444,260.280,-120.494,170.452,45.837,158.787
C03134=1029.451,260.529,-120.523,170.456,45.836,158.787
C03135=1029.457,260.777,-120.553,170.458,45.835,158.787
C03136=1029.465,261.025,-120.582,170.462,45.834,158.788
C03137=1029.471,261.273,-120.612,170.466,45.833,158.788
C03138=1029.477,261.522,-120.642,170.469,45.832,158.788
C03139=1029.484,261.769,-120.671,170.473,45.831,158.788
C03140=1029.491,262.018,-120.702,170.478,45.830,158.789
C03141=1029.497,262.266,-120.731,170.480,45.829,158.789
C03142=1029.504,262.514,-120.761,170.484,45.828,158.789
C03143=1029.514,262.886,-120.806,170.489,45.827,158.789
C03144=1029.524,263.258,-120.850,170.495,45.825,158.789
C03145=1029.534,263.630,-120.895,170.501,45.824,158.790
C03146=1029.543,264.002,-120.940,170.507,45.823,158.790
C03147=1029.550,264.250,-120.970,170.510,45.822,158.790
C03148=1029.557,264.498,-121.000,170.514,45.821,158.791
C03149=1029.564,264.746,-121.030,170.518,45.820,158.791
C03150=1029.570,264.995,-121.060,170.521,45.819,158.791
C03151=1029.577,265.242,-121.090,170.525,45.818,158.791
C03152=1029.584,265.491,-121.120,170.528,45.817,158.791
C03153=1029.590,265.739,-121.149,170.532,45.817,158.792
C03154=1029.597,265.987,-121.179,170.536,45.815,158.792
C03155=1029.604,266.235,-121.210,170.540,45.814,158.792
C03156=1029.610,266.483,-121.240,170.543,45.813,158.792
C03157=1029.618,266.731,-121.270,170.547,45.813,158.792
C03158=1029.623,266.979,-121.300,170.550,45.812,158.793
C03159=1029.631,267.227,-121.331,170.554,45.811,158.793
C03160=1029.638,267.475,-121.361,170.558,45.810,158.793
C03161=1029.644,267.723,-121.391,170.562,45.809,158.793
C03162=1029.651,267.971,-121.421,170.565,45.809,158.793
C03163=1029.657,268.220,-121.452,170.569,45.808,158.794
C03164=1029.664,268.467,-121.482,170.573,45.807,158.794
C03165=1029.671,268.716,-121.512,170.576,45.806,158.794
C03166=1029.677,268.964,-121.542,170.580,45.805,158.794
C03167=1029.684,269.212,-121.572,170.584,45.804,158.795
C03168=1029.691,269.460,-121.602,170.587,45.803,158.795
C03169=1029.697,269.708,-121.633,170.592,45.803,158.795
C03170=1029.704,269.956,-121.663,170.596,45.802,158.795
C03171=1029.710,270.204,-121.694,170.599,45.801,158.796
C03172=1029.718,270.453,-121.724,170.603,45.800,158.796
C03173=1029.723,270.700,-121.754,170.607,45.799,158.796
C03174=1029.731,270.948,-121.785,170.610,45.798,158.796
C03175=1029.737,271.196,-121.816,170.614,45.798,158.797
C03176=1029.744,271.444,-121.845,170.618,45.797,158.797
C03177=1029.750,271.693,-121.876,170.622,45.796,158.797
C03178=1029.757,271.941,-121.906,170.625,45.795,158.797
C03179=1029.764,272.189,-121.938,170.630,45.795,158.798
C03180=1029.771,272.436,-121.967,170.634,45.794,158.798
C03181=1029.777,272.685,-121.998,170.637,45.793,158.798
C03182=1029.784,272.932,-122.029,170.641,45.792,158.798
C03183=1029.791,273.181,-122.060,170.645,45.792,158.799
C03184=1029.797,273.429,-122.090,170.649,45.791,158.799
C03185=1029.804,273.677,-122.120,170.652,45.790,158.799
C03186=1029.811,273.925,-122.152,170.657,45.790,158.799
C03187=1029.818,274.173,-122.182,170.661,45.789,158.800
C03188=1029.824,274.420,-122.213,170.664,45.788,158.800
C03189=1029.830,274.669,-122.243,170.668,45.788,158.800
C03190=1029.837,274.917,-122.274,170.672,45.787,158.800
C03191=1029.844,275.165,-122.305,170.676,45.786,158.801
C03192=1029.851,275.413,-122.336,170.679,45.786,158.801
C03193=1029.857,275.660,-122.366,170.683,45.785,158.801
C03194=1029.864,275.909,-122.397,170.687,45.784,158.802
C03195=1029.871,276.157,-122.428,170.692,45.784,158.802
C03196=1029.878,276.405,-122.458,170.695,45.783,158.802
C03197=1029.885,276.653,-122.490,170.699,45.783,158.802
C03198=1029.891,276.901,-122.521,170.703,45.782,158.803
C03199=1029.901,277.277,-122.568,170.709,45.781,158.803
C03200=1029.912,277.654,-122.614,170.714,45.780,158.804
C03201=1029.922,278.031,-122.661,170.721,45.779,158.804
C03202=1029.932,278.407,-122.708,170.727,45.778,158.805
C03203=1029.938,278.656,-122.739,170.730,45.777,158.805
C03204=1029.945,278.903,-122.771,170.735,45.777,158.805
C03205=1029.952,279.151,-122.802,170.739,45.777,158.806
C03206=1029.958,279.399,-122.833,170.743,45.776,158.806
C03207=1029.965,279.648,-122.864,170.747,45.775,158.806
C03208=1029.972,279.895,-122.895,170.750,45.775,158.806
C03209=1029.979,280.143,-122.926,170.755,45.774,158.807
C03210=1029.986,280.391,-122.958,170.759,45.773,158.807
C03211=1029.992,280.640,-122.989,170.763,45.773,158.807
C03212=1029.998,280.887,-123.020,170.766,45.773,158.808
C03213=1030.005,281.135,-123.051,170.770,45.772,158.808
C03214=1030.012,281.383,-123.082,170.775,45.772,158.808
C03215=1030.018,281.631,-123.114,170.779,45.771,158.809
C03216=1030.025,281.879,-123.145,170.783,45.770,158.809
C03217=1030.031,282.127,-123.176,170.786,45.770,158.809
C03218=1030.039,282.375,-123.207,170.790,45.769,158.809
C03219=1030.046,282.623,-123.238,170.795,45.769,158.810
C03220=1030.052,282.870,-123.270,170.799,45.768,158.810
C03221=1030.059,283.118,-123.301,170.803,45.767,158.811
C03222=1030.066,283.366,-123.333,170.806,45.767,158.811
C03223=1030.073,283.614,-123.364,170.811,45.767,158.811
C03224=1030.079,283.862,-123.395,170.815,45.767,158.812
C03225=1030.086,284.110,-123.427,170.819,45.766,158.812
C03226=1030.093,284.358,-123.458,170.823,45.765,158.812
C03227=1030.099,284.606,-123.490,170.828,45.765,158.813
C03228=1030.106,284.854,-123.521,170.831,45.764,158.813
C03229=1030.114,285.101,-123.552,170.835,45.764,158.813
C03230=1030.121,285.350,-123.584,170.839,45.764,158.814
C03231=1030.128,285.598,-123.615,170.844,45.763,158.814
C03232=1030.134,285.846,-123.647,170.848,45.762,158.814
C03233=1030.141,286.094,-123.678,170.852,45.762,158.815
C03234=1030.148,286.341,-123.710,170.856,45.762,158.815
C03235=1030.155,286.589,-123.742,170.859,45.762,158.815
C03236=1030.161,286.837,-123.774,170.864,45.761,158.816
C03237=1030.168,287.085,-123.805,170.868,45.761,158.816
C03238=1030.174,287.333,-123.837,170.872,45.760,158.816
C03239=1030.181,287.580,-123.869,170.876,45.760,158.817
C03240=1030.188,287.828,-123.900,170.881,45.759,158.817
C03241=1030.195,288.076,-123.932,170.885,45.759,158.818
C03242=1030.202,288.324,-123.963,170.888,45.759,158.818
C03243=1030.209,288.572,-123.996,170.893,45.758,158.818
C03244=1030.215,288.820,-124.028,170.897,45.758,158.819
C03245=1030.222,289.068,-124.059,170.901,45.758,158.819
C03246=1030.229,289.315,-124.091,170.906,45.757,158.820
C03247=1030.236,289.563,-124.123,170.910,45.757,158.820
C03248=1030.243,289.810,-124.155,170.914,45.757,158.820
C03249=1030.249,290.059,-124.187,170.918,45.757,158.821
C03250=1030.256,290.307,-124.219,170.922,45.756,158.821
C03251=1030.263,290.554,-124.251,170.926,45.756,158.821
C03252=1030.270,290.802,-124.282,170.931,45.756,158.822
C03253=1030.276,291.050,-124.315,170.935,45.755,158.822
C03254=1030.283,291.299,-124.347,170.939,45.755,158.823
C03255=1030.293,291.687,-124.397,170.946,45.755,158.823
C03256=1030.305,292.076,-124.447,170.952,45.754,158.824
C03257=1030.316,292.465,-124.498,170.959,45.754,158.825
C03258=1030.326,292.854,-124.548,170.966,45.753,158.825
C03259=1030.333,293.101,-124.580,170.970,45.753,158.826
C03260=1030.340,293.349,-124.613,170.974,45.753,158.826
C03261=1030.347,293.597,-124.644,170.978,45.752,158.826
C03262=1030.354,293.844,-124.676,170.983,45.752,158.827
C03263=1030.361,294.093,-124.709,170.987,45.752,158.827
C03264=1030.367,294.341,-124.741,170.991,45.752,158.828
C03265=1030.374,294.588,-124.774,170.996,45.752,158.828
C03266=1030.381,294.835,-124.806,171.000,45.751,158.829
C03267=1030.387,295.084,-124.839,171.005,45.752,158.829
C03268=1030.394,295.331,-124.872,171.009,45.751,158.829
C03269=1030.400,295.579,-124.903,171.013,45.751,158.830
C03270=1030.407,295.827,-124.936,171.017,45.751,158.830
C03271=1030.414,296.075,-124.969,171.021,45.751,158.831
C03272=1030.421,296.322,-125.001,171.026,45.751,158.831
C03273=1030.427,296.570,-125.034,171.030,45.751,158.832
C03274=1030.434,296.818,-125.067,171.034,45.751,158.832
C03275=1030.441,297.066,-125.099,171.039,45.750,158.833
C03276=1030.447,297.313,-125.132,171.043,45.751,158.833
C03277=1030.453,297.561,-125.165,171.048,45.750,158.833
C03278=1030.461,297.809,-125.197,171.052,45.751,158.834
C03279=1030.467,298.056,-125.230,171.057,45.750,158.834
C03280=1030.474,298.304,-125.263,171.061,45.750,158.835
C03281=1030.481,298.552,-125.295,171.065,45.750,158.835
C03282=1030.488,298.800,-125.328,171.070,45.750,158.836
C03283=1030.495,299.048,-125.361,171.074,45.750,158.836
C03284=1030.501,299.295,-125.394,171.079,45.750,158.837
C03285=1030.508,299.542,-125.427,171.083,45.750,158.837
C03286=1030.515,299.790,-125.460,171.088,45.750,158.838
C03287=1030.521,300.038,-125.492,171.092,45.750,158.838
C03288=1030.529,300.286,-125.525,171.096,45.750,158.839
C03289=1030.535,300.534,-125.558,171.101,45.750,158.839
C03290=1030.542,300.782,-125.591,171.105,45.749,158.840
C03291=1030.550,301.028,-125.624,171.110,45.750,158.840
C03292=1030.556,301.276,-125.656,171.115,45.750,158.841
C03293=1030.563,301.524,-125.689,171.119,45.750,158.841
C03294=1030.569,301.772,-125.722,171.123,45.750,158.842
C03295=1030.577,302.019,-125.755,171.128,45.750,158.842
C03296=1030.583,302.267,-125.788,171.132,45.750,158.843
C03297=1030.590,302.515,-125.821,171.137,45.750,158.843
C03298=1030.597,302.762,-125.853,171.141,45.750,158.844
C03299=1030.604,303.010,-125.887,171.146,45.750,158.844
C03300=1030.611,303.258,-125.920,171.150,45.750,158.845
C03301=1030.618,303.506,-125.953,171.155,45.750,158.845
C03302=1030.625,303.753,-125.986,171.159,45.750,158.846
C03303=1030.632,304.001,-126.019,171.164,45.750,158.846
C03304=1030.639,304.249,-126.053,171.168,45.750,158.847
C03305=1030.645,304.496,-126.086,171.173,45.750,158.847
C03306=1030.653,304.744,-126.118,171.177,45.750,158.848
C03307=1030.660,304.992,-126.152,171.182,45.750,158.848
C03308=1030.666,305.240,-126.185,171.186,45.750,158.849
C03309=1030.674,305.487,-126.218,171.191,45.750,158.849
C03310=1030.681,305.734,-126.251,171.195,45.751,158.850
C03311=1030.692,306.140,-126.305,171.203,45.751,158.851
C03312=1030.704,306.546,-126.360,171.211,45.751,158.852
C03313=1030.716,306.952,-126.415,171.219,45.750,158.852
C03314=1030.727,307.359,-126.469,171.225,45.751,158.853
C03315=1030.734,307.606,-126.502,171.230,45.751,158.854
C03316=1030.741,307.853,-126.536,171.236,45.751,158.854
C03317=1030.749,308.101,-126.568,171.240,45.751,158.855
C03318=1030.756,308.349,-126.602,171.245,45.752,158.855
C03319=1030.763,308.596,-126.636,171.249,45.751,158.856
C03320=1030.769,308.844,-126.669,171.254,45.752,158.856
C03321=1030.777,309.092,-126.702,171.258,45.752,158.857
C03322=1030.785,309.339,-126.736,171.263,45.752,158.858
C03323=1030.791,309.587,-126.769,171.268,45.752,158.858
C03324=1030.798,309.835,-126.802,171.273,45.752,158.859
C03325=1030.805,310.082,-126.836,171.278,45.753,158.859
C03326=1030.813,310.330,-126.870,171.282,45.752,158.860
C03327=1030.820,310.577,-126.903,171.287,45.753,158.860
C03328=1030.827,310.825,-126.936,171.291,45.753,158.861
C03329=1030.834,311.073,-126.970,171.297,45.753,158.861
C03330=1030.841,311.320,-127.004,171.301,45.753,158.862
C03331=1030.848,311.568,-127.038,171.306,45.753,158.863
C03332=1030.855,311.815,-127.071,171.311,45.754,158.863
C03333=1030.861,312.063,-127.105,171.315,45.755,158.864
C03334=1030.869,312.310,-127.140,171.320,45.755,158.864
C03335=1030.876,312.558,-127.174,171.325,45.755,158.865
C03336=1030.882,312.805,-127.208,171.329,45.755,158.866
C03337=1030.889,313.053,-127.242,171.335,45.756,158.866
C03338=1030.896,313.300,-127.275,171.340,45.756,158.867
C03339=1030.903,313.548,-127.310,171.344,45.757,158.867
C03340=1030.910,313.795,-127.344,171.349,45.757,158.868
C03341=1030.917,314.043,-127.378,171.354,45.758,158.869
C03342=1030.923,314.290,-127.412,171.358,45.758,158.869
C03343=1030.931,314.538,-127.446,171.363,45.758,158.870
C03344=1030.937,314.785,-127.481,171.368,45.758,158.871
C03345=1030.945,315.033,-127.515,171.373,45.759,158.871
C03346=1030.952,315.281,-127.549,171.378,45.759,158.872
C03347=1030.958,315.529,-127.583,171.382,45.760,158.872
C03348=1030.966,315.776,-127.618,171.387,45.761,158.873
C03349=1030.973,316.023,-127.652,171.393,45.761,158.874
C03350=1030.979,316.271,-127.686,171.398,45.761,158.875
C03351=1030.986,316.518,-127.720,171.402,45.762,158.875
C03352=1030.993,316.766,-127.755,171.407,45.762,158.876
C03353=1031.000,317.013,-127.789,171.412,45.763,158.876
C03354=1031.007,317.260,-127.823,171.417,45.763,158.877
C03355=1031.014,317.508,-127.858,171.422,45.763,158.878
C03356=1031.021,317.756,-127.892,171.427,45.764,158.878
C03357=1031.028,318.003,-127.927,171.431,45.764,158.879
C03358=1031.035,318.251,-127.961,171.436,45.765,158.880
C03359=1031.043,318.498,-127.996,171.442,45.765,158.880
C03360=1031.049,318.746,-128.030,171.447,45.766,158.881
C03361=1031.057,318.993,-128.065,171.451,45.766,158.882
C03362=1031.064,319.241,-128.099,171.456,45.767,158.882
C03363=1031.071,319.488,-128.134,171.462,45.767,158.883
C03364=1031.079,319.736,-128.168,171.467,45.768,158.884
C03365=1031.085,319.983,-128.203,171.471,45.768,158.884
C03366=1031.093,320.230,-128.237,171.477,45.769,158.885
C03367=1031.105,320.642,-128.294,171.485,45.770,158.886
C03368=1031.116,321.053,-128.351,171.493,45.770,158.887
C03369=1031.129,321.464,-128.409,171.502,45.772,158.888
C03370=1031.140,321.874,-128.468,171.510,45.773,158.889
C03371=1031.148,322.122,-128.502,171.515,45.773,158.890
C03372=1031.155,322.369,-128.536,171.521,45.773,158.891
C03373=1031.162,322.616,-128.571,171.525,45.774,158.892
C03374=1031.169,322.863,-128.606,171.530,45.775,158.892
C03375=1031.176,323.112,-128.641,171.536,45.775,158.893
C03376=1031.184,323.359,-128.675,171.541,45.776,158.894
C03377=1031.191,323.607,-128.710,171.546,45.777,158.894
C03378=1031.198,323.854,-128.745,171.551,45.777,158.895
C03379=1031.206,324.101,-128.780,171.556,45.778,158.896
C03380=1031.213,324.349,-128.815,171.561,45.779,158.896
C03381=1031.221,324.596,-128.849,171.567,45.779,158.897
C03382=1031.228,324.844,-128.885,171.571,45.780,158.898
C03383=1031.235,325.091,-128.919,171.577,45.780,158.899
C03384=1031.242,325.338,-128.955,171.582,45.781,158.899
C03385=1031.250,325.586,-128.990,171.587,45.782,158.900
C03386=1031.257,325.833,-129.025,171.593,45.783,158.901
C03387=1031.265,326.080,-129.059,171.597,45.783,158.901
C03388=1031.273,326.328,-129.094,171.603,45.783,158.902
C03389=1031.280,326.576,-129.129,171.608,45.784,158.903
C03390=1031.288,326.823,-129.164,171.613,45.785,158.904
C03391=1031.294,327.071,-129.199,171.619,45.786,158.905
C03392=1031.302,327.318,-129.234,171.624,45.787,158.905
C03393=1031.309,327.566,-129.269,171.630,45.787,158.906
C03394=1031.317,327.813,-129.304,171.634,45.787,158.907
C03395=1031.324,328.060,-129.340,171.640,45.788,158.907
C03396=1031.331,328.308,-129.375,171.645,45.790,158.908
C03397=1031.338,328.555,-129.410,171.650,45.790,158.909
C03398=1031.346,328.802,-129.447,171.656,45.791,158.910
C03399=1031.353,329.050,-129.481,171.661,45.792,158.911
C03400=1031.361,329.298,-129.517,171.667,45.793,158.911
C03401=1031.368,329.544,-129.552,171.672,45.793,158.912
C03402=1031.375,329.792,-129.588,171.676,45.794,158.913
C03403=1031.382,330.039,-129.624,171.683,45.795,158.914
C03404=1031.389,330.287,-129.659,171.687,45.796,158.915
C03405=1031.396,330.534,-129.695,171.693,45.797,158.915
C03406=1031.404,330.782,-129.731,171.698,45.798,158.916
C03407=1031.412,331.028,-129.766,171.704,45.798,158.917
C03408=1031.419,331.277,-129.801,171.709,45.800,158.918
C03409=1031.426,331.523,-129.837,171.715,45.800,158.919
C03410=1031.433,331.771,-129.873,171.720,45.801,158.919
C03411=1031.441,332.018,-129.909,171.726,45.802,158.920
C03412=1031.448,332.266,-129.945,171.731,45.803,158.921
C03413=1031.455,332.513,-129.980,171.736,45.804,158.922
C03414=1031.463,332.760,-130.016,171.742,45.805,158.923
C03415=1031.470,333.008,-130.052,171.747,45.806,158.923
C03416=1031.477,333.255,-130.088,171.753,45.807,158.924
C03417=1031.486,333.502,-130.123,171.759,45.808,158.925
C03418=1031.493,333.749,-130.159,171.764,45.809,158.926
C03419=1031.500,333.996,-130.195,171.770,45.810,158.927
C03420=1031.508,334.245,-130.231,171.775,45.810,158.928
C03421=1031.515,334.491,-130.267,171.781,45.812,158.928
C03422=1031.522,334.739,-130.303,171.786,45.813,158.929
C03423=1031.534,335.145,-130.362,171.795,45.814,158.931
C03424=1031.546,335.551,-130.422,171.804,45.816,158.932
C03425=1031.559,335.958,-130.481,171.813,45.818,158.934
C03426=1031.571,336.364,-130.541,171.822,45.820,158.935
C03427=1031.578,336.612,-130.577,171.828,45.821,158.936
C03428=1031.585,336.858,-130.613,171.833,45.822,158.937
C03429=1031.592,337.106,-130.649,171.840,45.823,158.938
C03430=1031.600,337.354,-130.686,171.844,45.824,158.938
C03431=1031.608,337.600,-130.723,171.851,45.825,158.939
C03432=1031.615,337.847,-130.758,171.856,45.827,158.940
C03433=1031.623,338.095,-130.795,171.862,45.827,158.941
C03434=1031.630,338.342,-130.831,171.867,45.829,158.942
C03435=1031.637,338.590,-130.868,171.873,45.830,158.943
C03436=1031.645,338.837,-130.904,171.879,45.831,158.944
C03437=1031.652,339.083,-130.940,171.884,45.832,158.945
C03438=1031.660,339.331,-130.977,171.890,45.833,158.946
C03439=1031.668,339.578,-131.013,171.896,45.834,158.947
C03440=1031.676,339.825,-131.050,171.901,45.836,158.948
C03441=1031.683,340.073,-131.087,171.908,45.837,158.949
C03442=1031.690,340.320,-131.123,171.912,45.838,158.949
C03443=1031.698,340.567,-131.160,171.919,45.839,158.950
C03444=1031.706,340.815,-131.196,171.925,45.840,158.951
C03445=1031.712,341.062,-131.232,171.930,45.842,158.952
C03446=1031.720,341.308,-131.269,171.936,45.843,158.953
C03447=1031.728,341.556,-131.306,171.942,45.844,158.954
C03448=1031.735,341.803,-131.343,171.947,45.846,158.955
C03449=1031.743,342.050,-131.379,171.954,45.847,158.956
C03450=1031.750,342.298,-131.417,171.960,45.848,158.957
C03451=1031.758,342.544,-131.454,171.965,45.849,158.958
C03452=1031.765,342.792,-131.491,171.971,45.851,158.959
C03453=1031.773,343.039,-131.528,171.977,45.852,158.960
C03454=1031.781,343.286,-131.564,171.982,45.853,158.961
C03455=1031.788,343.534,-131.601,171.989,45.855,158.962
C03456=1031.796,343.780,-131.638,171.995,45.856,158.963
C03457=1031.803,344.028,-131.676,172.000,45.858,158.964
C03458=1031.811,344.275,-131.712,172.006,45.859,158.965
C03459=1031.818,344.522,-131.750,172.012,45.860,158.966
C03460=1031.826,344.769,-131.786,172.019,45.861,158.967
C03461=1031.833,345.016,-131.824,172.024,45.863,158.968
C03462=1031.841,345.263,-131.861,172.030,45.864,158.969
C03463=1031.849,345.510,-131.898,172.036,45.866,158.970
C03464=1031.856,345.757,-131.935,172.042,45.867,158.971
C03465=1031.864,346.005,-131.972,172.048,45.869,158.972
C03466=1031.872,346.252,-132.009,172.054,45.870,158.973
C03467=1031.879,346.499,-132.047,172.060,45.871,158.974
C03468=1031.887,346.746,-132.084,172.067,45.873,158.975
C03469=1031.895,346.993,-132.121,172.072,45.874,158.976
C03470=1031.903,347.240,-132.158,172.078,45.876,158.977
C03471=1031.910,347.487,-132.196,172.084,45.877,158.978
C03472=1031.918,347.735,-132.233,172.091,45.879,158.979
C03473=1031.926,347.982,-132.271,172.097,45.880,158.980
C03474=1031.934,348.229,-132.308,172.102,45.882,158.981
C03475=1031.941,348.475,-132.346,172.109,45.884,158.982
C03476=1031.948,348.722,-132.383,172.115,45.885,158.983
C03477=1031.957,348.970,-132.421,172.121,45.887,158.984
C03478=1031.964,349.217,-132.458,172.127,45.888,158.985
C03479=1031.976,349.620,-132.520,172.138,45.891,158.987
C03480=1031.990,350.023,-132.581,172.147,45.893,158.989
C03481=1032.002,350.426,-132.643,172.157,45.896,158.991
C03482=1032.015,350.829,-132.704,172.167,45.898,158.992
C03483=1032.022,351.076,-132.743,172.173,45.900,158.993
C03484=1032.030,351.323,-132.780,172.180,45.902,158.994
C03485=1032.038,351.570,-132.819,172.186,45.904,158.996
C03486=1032.046,351.817,-132.856,172.192,45.905,158.997
C03487=1032.053,352.063,-132.894,172.199,45.907,158.998
C03488=1032.061,352.311,-132.932,172.205,45.908,158.999
C03489=1032.069,352.558,-132.970,172.211,45.910,159.000
C03490=1032.077,352.806,-133.008,172.217,45.912,159.001
C03491=1032.085,353.052,-133.046,172.224,45.914,159.002
C03492=1032.092,353.299,-133.083,172.230,45.915,159.003
C03493=1032.100,353.546,-133.122,172.236,45.917,159.004
C03494=1032.108,353.793,-133.160,172.243,45.919,159.006
C03495=1032.116,354.040,-133.198,172.249,45.920,159.007
C03496=1032.124,354.287,-133.235,172.256,45.922,159.008
C03497=1032.132,354.534,-133.274,172.262,45.924,159.009
C03498=1032.140,354.780,-133.312,172.269,45.926,159.010
C03499=1032.148,355.028,-133.351,172.275,45.927,159.011
C03500=1032.155,355.275,-133.388,172.281,45.929,159.013
C03501=1032.164,355.522,-133.426,172.288,45.931,159.014
C03502=1032.171,355.768,-133.465,172.294,45.933,159.015
C03503=1032.180,356.015,-133.503,172.301,45.934,159.016
C03504=1032.188,356.263,-133.542,172.307,45.936,159.017
C03505=1032.195,356.509,-133.580,172.314,45.939,159.018
C03506=1032.203,356.756,-133.619,172.320,45.940,159.020
C03507=1032.211,357.003,-133.657,172.327,45.942,159.021
C03508=1032.219,357.250,-133.696,172.333,45.944,159.022
C03509=1032.227,357.497,-133.734,172.340,45.946,159.023
C03510=1032.235,357.744,-133.773,172.346,45.948,159.024
C03511=1032.243,357.991,-133.811,172.353,45.950,159.026
C03512=1032.250,358.237,-133.851,172.359,45.951,159.027
C03513=1032.258,358.484,-133.889,172.366,45.954,159.028
C03514=1032.266,358.732,-133.928,172.373,45.956,159.029
C03515=1032.274,358.978,-133.966,172.379,45.957,159.030
C03516=1032.282,359.225,-134.005,172.386,45.960,159.032
C03517=1032.291,359.472,-134.044,172.392,45.961,159.033
C03518=1032.299,359.719,-134.083,172.400,45.964,159.034
C03519=1032.306,359.966,-134.121,172.406,45.965,159.035
C03520=1032.315,360.212,-134.160,172.413,45.967,159.037
C03521=1032.323,360.459,-134.199,172.420,45.969,159.038
C03522=1032.331,360.706,-134.238,172.426,45.971,159.039
C03523=1032.339,360.953,-134.276,172.433,45.974,159.040
C03524=1032.347,361.200,-134.315,172.440,45.976,159.042
C03525=1032.355,361.447,-134.355,172.446,45.978,159.043
C03526=1032.363,361.693,-134.394,172.454,45.980,159.044
C03527=1032.371,361.941,-134.433,172.460,45.982,159.046
C03528=1032.378,362.187,-134.472,172.467,45.984,159.047
C03529=1032.387,362.434,-134.511,172.474,45.986,159.048
C03530=1032.395,362.681,-134.550,172.480,45.988,159.049
C03531=1032.403,362.927,-134.590,172.487,45.991,159.051
C03532=1032.411,363.174,-134.630,172.495,45.992,159.052
C03533=1032.419,363.421,-134.668,172.501,45.995,159.053
C03534=1032.427,363.667,-134.708,172.508,45.997,159.055
C03535=1032.440,364.077,-134.773,172.520,46.001,159.057
C03536=1032.454,364.486,-134.838,172.531,46.004,159.059
C03537=1032.468,364.896,-134.904,172.542,46.008,159.061
C03538=1032.481,365.304,-134.970,172.554,46.011,159.063
C03539=1032.490,365.551,-135.009,172.561,46.014,159.065
C03540=1032.498,365.798,-135.049,172.568,46.016,159.066
C03541=1032.506,366.045,-135.088,172.575,46.018,159.068
C03542=1032.514,366.291,-135.128,172.582,46.020,159.069
C03543=1032.522,366.538,-135.167,172.589,46.023,159.070
C03544=1032.531,366.785,-135.207,172.596,46.025,159.072
C03545=1032.538,367.032,-135.247,172.604,46.028,159.073
C03546=1032.547,367.278,-135.286,172.611,46.030,159.074
C03547=1032.555,367.525,-135.325,172.617,46.032,159.076
C03548=1032.564,367.772,-135.366,172.625,46.035,159.077
C03549=1032.572,368.018,-135.406,172.632,46.037,159.079
C03550=1032.581,368.265,-135.445,172.639,46.039,159.080
C03551=1032.589,368.512,-135.485,172.647,46.042,159.081
C03552=1032.597,368.758,-135.525,172.653,46.044,159.083
C03553=1032.605,369.005,-135.565,172.660,46.046,159.084
C03554=1032.614,369.252,-135.604,172.668,46.049,159.086
C03555=1032.623,369.498,-135.645,172.675,46.051,159.087
C03556=1032.631,369.745,-135.684,172.683,46.053,159.088
C03557=1032.639,369.991,-135.725,172.690,46.056,159.090
C03558=1032.648,370.238,-135.765,172.696,46.059,159.091
C03559=1032.656,370.485,-135.805,172.705,46.061,159.093
C03560=1032.663,370.732,-135.845,172.711,46.064,159.094
C03561=1032.672,370.978,-135.885,172.719,46.066,159.096
C03562=1032.680,371.224,-135.926,172.726,46.069,159.097
C03563=1032.689,371.471,-135.966,172.733,46.071,159.099
C03564=1032.697,371.717,-136.006,172.741,46.074,159.100
C03565=1032.705,371.964,-136.047,172.748,46.076,159.102
C03566=1032.714,372.211,-136.088,172.756,46.079,159.103
C03567=1032.722,372.457,-136.129,172.763,46.082,159.105
C03568=1032.730,372.704,-136.168,172.771,46.085,159.106
C03569=1032.739,372.951,-136.209,172.778,46.087,159.108
C03570=1032.747,373.197,-136.250,172.786,46.089,159.109
C03571=1032.756,373.443,-136.290,172.793,46.092,159.111
C03572=1032.765,373.690,-136.331,172.801,46.095,159.112
C03573=1032.773,373.936,-136.371,172.808,46.098,159.114
C03574=1032.782,374.183,-136.412,172.816,46.100,159.115
C03575=1032.790,374.429,-136.452,172.823,46.103,159.117
C03576=1032.799,374.676,-136.493,172.831,46.105,159.118
C03577=1032.807,374.922,-136.534,172.839,46.108,159.120
C03578=1032.816,375.169,-136.574,172.846,46.111,159.122
C03579=1032.824,375.415,-136.615,172.854,46.114,159.123
C03580=1032.833,375.662,-136.656,172.861,46.116,159.125
C03581=1032.842,375.908,-136.697,172.869,46.119,159.126
C03582=1032.850,376.155,-136.738,172.877,46.122,159.128
C03583=1032.858,376.401,-136.778,172.884,46.124,159.129
C03584=1032.867,376.648,-136.819,172.893,46.128,159.131
C03585=1032.877,376.894,-136.860,172.901,46.130,159.133
C03586=1032.885,377.140,-136.901,172.908,46.133,159.134
C03587=1032.893,377.387,-136.942,172.916,46.136,159.136
C03588=1032.902,377.634,-136.984,172.924,46.138,159.137
C03589=1032.911,377.880,-137.024,172.931,46.141,159.139
C03590=1032.920,378.126,-137.066,172.939,46.144,159.141
C03591=1032.927,378.344,-137.102,172.946,46.147,159.142
C03592=1032.935,378.562,-137.138,172.953,46.150,159.144
C03593=1032.942,378.780,-137.175,172.960,46.152,159.145
C03594=1032.950,378.997,-137.212,172.967,46.155,159.146
C03595=1032.958,379.215,-137.249,172.974,46.158,159.148
